  MoveL 782 to (-960, 800, -0.5) mm, rotated rx -180 ry 0 rz 90 deg; joints [11.922, -75.22, 120.913, -51.827, 9.519, 60.758]
  MoveL 783 to (-960, 800, 50) mm, rotated rx 180 ry 0 rz 90 deg; joints [11.922, -77.377, 120.292, -40.937, 11.444, 49.686]
  MoveL 784 to (-960, 850, 50) mm, rotated rx -180 ry 0 rz 90 deg; joints [12.344, -79.438, 122.916, -43.67, 11.235, 52.769]
  MoveL 785 to (-960, 850, -0.5) mm, rotated rx -180 ry 0 rz 90 deg; joints [12.344, -77.191, 123.556, -55.829, 9.358, 65.123]
  MoveL 786 to (-960, 850, 50) mm, rotated rx -180 ry 0 rz 90 deg; joints [12.344, -79.438, 122.916, -43.67, 11.235, 52.769]
  MoveL 787 to (-960, 900, 50) mm, rotated rx 180 ry 0 rz 90 deg; joints [12.796, -81.543, 125.497, -46.231, 11.128, 55.698]
  MoveL 788 to (-960, 900, -0.5) mm, rotated rx 180 ry 0 rz 90 deg; joints [12.796, -79.199, 126.159, -59.572, 9.302, 69.249]
  MoveL 789 to (-960, 900, 50) mm, rotated rx 180 ry 0 rz 90 deg; joints [12.796, -81.543, 125.497, -46.231, 11.128, 55.698]
  MoveL 790 to (-960, 950, 50) mm, rotated rx 180 ry 0 rz 90 deg; joints [13.282, -83.7, 128.037, -48.525, 11.126, 58.38]
  MoveL 791 to (-960, 950, -0.5) mm, rotated rx -180 ry 0 rz 90 deg; joints [13.282, -81.252, 128.723, -62.909, 9.346, 72.993]
  MoveL 792 to (-960, 950, 50) mm, rotated rx 180 ry 0 rz 90 deg; joints [13.282, -83.7, 128.037, -48.525, 11.126, 58.38]
  MoveL 793 to (-960, 1000, 50) mm, rotated rx 180 ry 0 rz 90 deg; joints [13.805, -85.92, 130.536, -50.46, 11.229, 60.727]
  MoveL 794 to (-960, 1000, -0.5) mm, rotated rx -180 ry 0 rz 90 deg; joints [13.805, -83.361, 131.25, -65.713, 9.483, 76.227]
  MoveL 795 to (-960, 1000, 50) mm, rotated rx 180 ry 0 rz 90 deg; joints [13.805, -85.92, 130.536, -50.46, 11.229, 60.727]
  MoveL 796 to (-960, 1050, 50) mm, rotated rx 180 ry 0 rz 90 deg; joints [14.371, -88.215, 132.994, -51.956, 11.439, 62.658]
  MoveL 797 to (-960, 1050, -0.5) mm, rotated rx 180 ry 0 rz 90 deg; joints [14.371, -85.537, 133.739, -67.879, 9.707, 78.851]
  MoveL 798 to (-960, 1050, 50) mm, rotated rx 180 ry 0 rz 90 deg; joints [14.371, -88.215, 132.994, -51.956, 11.439, 62.658]
  MoveL 799 to (-960, 1100, 50) mm, rotated rx 180 ry 0 rz 90 deg; joints [14.983, -90.599, 135.413, -52.948, 11.763, 64.112]
  MoveL 800 to (-960, 1100, -0.5) mm, rotated rx 180 ry 0 rz 90 deg; joints [14.983, -87.793, 136.192, -69.331, 10.015, 80.788]
  MoveL 801 to (-960, 1100, 50) mm, rotated rx 180 ry 0 rz 90 deg; joints [14.983, -90.599, 135.413, -52.948, 11.763, 64.112]
  MoveL 802 to (-960, 1150, 50) mm, rotated rx 180 ry 0 rz 90 deg; joints [15.649, -93.088, 137.79, -53.393, 12.209, 65.046]
  MoveL 803 to (-960, 1150, -0.5) mm, rotated rx 180 ry 0 rz 90 deg; joints [15.649, -90.145, 138.607, -70.016, 10.407, 81.99]
  MoveL 804 to (-960, 1150, 50) mm, rotated rx 180 ry 0 rz 90 deg; joints [15.649, -93.088, 137.79, -53.393, 12.209, 65.046]
  MoveL 805 to (-960, 1200, 50) mm, rotated rx 180 ry 0 rz 90 deg; joints [16.376, -95.702, 140.125, -53.269, 12.79, 65.44]
  MoveL 806 to (-960, 1200, -0.5) mm, rotated rx 180 ry 0 rz 90 deg; joints [16.376, -92.612, 140.985, -69.905, 10.89, 82.431]
  MoveL 807 to (-960, 1200, 50) mm, rotated rx 180 ry 0 rz 90 deg; joints [16.376, -95.702, 140.125, -53.269, 12.79, 65.44]
  MoveL 808 to (-960, 1250, 50) mm, rotated rx 180 ry 0 rz 90 deg; joints [17.171, -98.462, 142.415, -52.579, 13.529, 65.301]
  MoveL 809 to (-960, 1250, -0.5) mm, rotated rx 180 ry 0 rz 90 deg; joints [17.171, -95.217, 143.324, -68.993, 11.479, 82.105]
  MoveL 810 to (-960, 1250, 50) mm, rotated rx 180 ry 0 rz 90 deg; joints [17.171, -98.462, 142.415, -52.579, 13.529, 65.301]
  MoveL 811 to (-960, 1300, 50) mm, rotated rx -180 ry 0 rz 90 deg; joints [18.044, -101.397, 144.658, -51.352, 14.453, 64.657]
  MoveL 812 to (-960, 1300, -0.5) mm, rotated rx -180 ry 0 rz 90 deg; joints [18.044, -97.987, 145.622, -67.292, 12.199, 81.029]
  MoveL 813 to (-960, 1300, 50) mm, rotated rx -180 ry 0 rz 90 deg; joints [18.044, -101.397, 144.658, -51.352, 14.453, 64.657]
  MoveL 814 to (-960, 1350, 50) mm, rotated rx -180 ry 0 rz 90 deg; joints [19.007, -104.538, 146.849, -49.641, 15.603, 63.564]
  MoveL 815 to (-960, 1350, -0.5) mm, rotated rx 180 ry 0 rz 90 deg; joints [19.007, -100.957, 147.875, -64.845, 13.087, 79.247]
  MoveL 816 to (-960, 1350, 50) mm, rotated rx -180 ry 0 rz 90 deg; joints [19.007, -104.538, 146.849, -49.641, 15.603, 63.564]
  MoveL 817 to (-960, 1400, 50) mm, rotated rx -180 ry 0 rz 90 deg; joints [20.075, -107.924, 148.982, -47.525, 17.03, 62.099]
  MoveL 818 to (-960, 1400, -0.5) mm, rotated rx -180 ry 0 rz 90 deg; joints [20.075, -104.168, 150.079, -61.73, 14.198, 76.837]
  MoveL 819 to (-960, 1400, 50) mm, rotated rx -180 ry 0 rz 90 deg; joints [20.075, -107.924, 148.982, -47.525, 17.03, 62.099]
  MoveL 820 to (-960, 1450, 50) mm, rotated rx -180 ry 0 rz 90 deg; joints [21.264, -111.599, 151.05, -45.102, 18.795, 60.359]
  MoveL 821 to (-960, 1450, -0.5) mm, rotated rx 180 ry 0 rz 90 deg; joints [21.264, -107.67, 152.227, -58.062, 15.601, 73.915]
  MoveL 822 to (-960, 1450, 50) mm, rotated rx -180 ry 0 rz 90 deg; joints [21.264, -111.599, 151.05, -45.102, 18.795, 60.359]
  MoveL 823 to (-1030, 50, 50) mm, rotated rx 180 ry 0 rz 90 deg; joints [9.672, -46.591, 72.453, -13.855, 26.202, 20.023]
  MoveL 824 to (-1030, 50, -0.5) mm, rotated rx -180 ry 0 rz 90 deg; joints [9.672, -45.337, 72.996, -14.794, 24.462, 21.062]
  MoveL 825 to (-1030, 50, 50) mm, rotated rx 180 ry 0 rz 90 deg; joints [9.672, -46.591, 72.453, -13.855, 26.202, 20.023]
  MoveL 826 to (-1030, 100, 50) mm, rotated rx 180 ry 0 rz 90 deg; joints [9.896, -48.808, 76.299, -15.015, 24.675, 21.419]
  MoveL 827 to (-1030, 100, -0.5) mm, rotated rx -180 ry 0 rz 90 deg; joints [9.896, -47.51, 76.834, -16.131, 22.91, 22.638]
  MoveL 828 to (-1030, 100, 50) mm, rotated rx 180 ry 0 rz 90 deg; joints [9.896, -48.808, 76.299, -15.015, 24.675, 21.419]
  MoveL 829 to (-1030, 150, 50) mm, rotated rx 180 ry 0 rz 90 deg; joints [10.13, -50.96, 79.988, -16.284, 23.25, 22.928]
  MoveL 830 to (-1030, 150, -0.5) mm, rotated rx 180 ry 0 rz 90 deg; joints [10.13, -49.618, 80.517, -17.61, 21.46, 24.362]
  MoveL 831 to (-1030, 150, 50) mm, rotated rx 180 ry 0 rz 90 deg; joints [10.13, -50.96, 79.988, -16.284, 23.25, 22.928]
  MoveL 832 to (-1030, 200, 50) mm, rotated rx 180 ry 0 rz 90 deg; joints [10.375, -53.058, 83.54, -17.672, 21.922, 24.564]
  MoveL 833 to (-1030, 200, -0.5) mm, rotated rx 180 ry 0 rz 90 deg; joints [10.375, -51.67, 84.065, -19.25, 20.106, 26.254]
  MoveL 834 to (-1030, 200, 50) mm, rotated rx 180 ry 0 rz 90 deg; joints [10.375, -53.058, 83.54, -17.672, 21.922, 24.564]
  MoveL 835 to (-1030, 250, 50) mm, rotated rx 180 ry 0 rz 90 deg; joints [10.632, -55.112, 86.972, -19.192, 20.684, 26.338]
  MoveL 836 to (-1030, 250, -0.5) mm, rotated rx -180 ry 0 rz 90 deg; joints [10.632, -53.676, 87.495, -21.069, 18.844, 28.332]
  MoveL 837 to (-1030, 250, 50) mm, rotated rx 180 ry 0 rz 90 deg; joints [10.632, -55.112, 86.972, -19.192, 20.684, 26.338]
  MoveL 838 to (-1030, 300, 50) mm, rotated rx 180 ry 0 rz 90 deg; joints [10.903, -57.13, 90.296, -20.854, 19.534, 28.262]
  MoveL 839 to (-1030, 300, -0.5) mm, rotated rx -180 ry 0 rz 90 deg; joints [10.903, -55.645, 90.82, -23.087, 17.671, 30.618]
  MoveL 840 to (-1030, 300, 50) mm, rotated rx 180 ry 0 rz 90 deg; joints [10.903, -57.13, 90.296, -20.854, 19.534, 28.262]
  MoveL 841 to (-1030, 350, 50) mm, rotated rx -180 ry 0 rz 90 deg; joints [11.187, -59.119, 93.525, -22.667, 18.471, 30.347]
  MoveL 842 to (-1030, 350, -0.5) mm, rotated rx 180 ry 0 rz 90 deg; joints [11.187, -57.583, 94.051, -25.322, 16.586, 33.131]
  MoveL 843 to (-1030, 350, 50) mm, rotated rx -180 ry 0 rz 90 deg; joints [11.187, -59.119, 93.525, -22.667, 18.471, 30.347]
  MoveL 844 to (-1030, 400, 50) mm, rotated rx -180 ry 0 rz 90 deg; joints [11.486, -61.086, 96.667, -24.639, 17.492, 32.601]
  MoveL 845 to (-1030, 400, -0.5) mm, rotated rx 180 ry 0 rz 90 deg; joints [11.486, -59.497, 97.197, -27.791, 15.591, 35.888]
  MoveL 846 to (-1030, 400, 50) mm, rotated rx -180 ry 0 rz 90 deg; joints [11.486, -61.086, 96.667, -24.639, 17.492, 32.601]
  MoveL 847 to (-1030, 450, 50) mm, rotated rx -180 ry 0 rz 90 deg; joints [11.801, -63.037, 99.73, -26.776, 16.601, 35.03]
  MoveL 848 to (-1030, 450, -0.5) mm, rotated rx -180 ry 0 rz 90 deg; joints [11.801, -61.393, 100.265, -30.507, 14.687, 38.904]
  MoveL 849 to (-1030, 450, 50) mm, rotated rx -180 ry 0 rz 90 deg; joints [11.801, -63.037, 99.73, -26.776, 16.601, 35.03]
  MoveL 850 to (-1030, 500, 50) mm, rotated rx 180 ry 0 rz 90 deg; joints [12.134, -64.977, 102.721, -29.075, 15.796, 37.633]
  MoveL 851 to (-1030, 500, -0.5) mm, rotated rx 180 ry 0 rz 90 deg; joints [12.134, -63.275, 103.263, -33.475, 13.876, 42.184]
  MoveL 852 to (-1030, 500, 50) mm, rotated rx 180 ry 0 rz 90 deg; joints [12.134, -64.977, 102.721, -29.075, 15.796, 37.633]
  MoveL 853 to (-1030, 550, 50) mm, rotated rx 180 ry 0 rz 90 deg; joints [12.486, -66.913, 105.646, -31.528, 15.081, 40.405]
  MoveL 854 to (-1030, 550, -0.5) mm, rotated rx 180 ry 0 rz 90 deg; joints [12.486, -65.149, 106.196, -36.688, 13.163, 45.724]
  MoveL 855 to (-1030, 550, 50) mm, rotated rx 180 ry 0 rz 90 deg; joints [12.486, -66.913, 105.646, -31.528, 15.081, 40.405]
  MoveL 856 to (-1030, 600, 50) mm, rotated rx 180 ry 0 rz 90 deg; joints [12.858, -68.849, 108.509, -34.12, 14.458, 43.328]
  MoveL 857 to (-1030, 600, -0.5) mm, rotated rx 180 ry 0 rz 90 deg; joints [12.858, -67.02, 109.069, -40.125, 12.551, 49.503]
  MoveL 858 to (-1030, 600, 50) mm, rotated rx 180 ry 0 rz 90 deg; joints [12.858, -68.849, 108.509, -34.12, 14.458, 43.328]
  MoveL 859 to (-1030, 650, 50) mm, rotated rx 180 ry 0 rz 90 deg; joints [13.253, -70.791, 111.315, -36.821, 13.93, 46.377]
  MoveL 860 to (-1030, 650, -0.5) mm, rotated rx 180 ry 0 rz 90 deg; joints [13.253, -68.894, 111.886, -43.746, 12.044, 53.482]
  MoveL 861 to (-1030, 650, 50) mm, rotated rx 180 ry 0 rz 90 deg; joints [13.253, -70.791, 111.315, -36.821, 13.93, 46.377]
  MoveL 862 to (-1030, 700, 50) mm, rotated rx 180 ry 0 rz 90 deg; joints [13.673, -72.744, 114.067, -39.592, 13.498, 49.512]
  MoveL 863 to (-1030, 700, -0.5) mm, rotated rx 180 ry 0 rz 90 deg; joints [13.673, -70.774, 114.651, -47.488, 11.643, 57.6]
  MoveL 864 to (-1030, 700, 50) mm, rotated rx 180 ry 0 rz 90 deg; joints [13.673, -72.744, 114.067, -39.592, 13.498, 49.512]
  MoveL 865 to (-1030, 750, 50) mm, rotated rx 180 ry 0 rz 90 deg; joints [14.12, -74.715, 116.768, -42.38, 13.165, 52.682]
  MoveL 866 to (-1030, 750, -0.5) mm, rotated rx -180 ry 0 rz 90 deg; joints [14.12, -72.668, 117.367, -51.27, 11.35, 61.777]
  MoveL 867 to (-1030, 750, 50) mm, rotated rx 180 ry 0 rz 90 deg; joints [14.12, -74.715, 116.768, -42.38, 13.165, 52.682]
  MoveL 868 to (-1030, 800, 50) mm, rotated rx 180 ry 0 rz 90 deg; joints [14.596, -76.709, 119.421, -45.122, 12.932, 55.826]
  MoveL 869 to (-1030, 800, -0.5) mm, rotated rx -180 ry 0 rz 90 deg; joints [14.596, -74.58, 120.037, -54.992, 11.164, 65.916]
  MoveL 870 to (-1030, 800, 50) mm, rotated rx 180 ry 0 rz 90 deg; joints [14.596, -76.709, 119.421, -45.122, 12.932, 55.826]
  MoveL 871 to (-1030, 850, 50) mm, rotated rx 180 ry 0 rz 90 deg; joints [15.104, -78.733, 122.029, -47.746, 12.8, 58.873]
  MoveL 872 to (-1030, 850, -0.5) mm, rotated rx 180 ry 0 rz 90 deg; joints [15.104, -76.517, 122.662, -58.546, 11.083, 69.91]
  MoveL 873 to (-1030, 850, 50) mm, rotated rx 180 ry 0 rz 90 deg; joints [15.104, -78.733, 122.029, -47.746, 12.8, 58.873]
  MoveL 874 to (-1030, 900, 50) mm, rotated rx 180 ry 0 rz 90 deg; joints [15.648, -80.795, 124.591, -50.177, 12.769, 61.751]
  MoveL 875 to (-1030, 900, -0.5) mm, rotated rx 180 ry 0 rz 90 deg; joints [15.648, -78.486, 125.246, -61.823, 11.103, 73.651]
  MoveL 876 to (-1030, 900, 50) mm, rotated rx 180 ry 0 rz 90 deg; joints [15.648, -80.795, 124.591, -50.177, 12.769, 61.751]
  MoveL 877 to (-1030, 950, 50) mm, rotated rx -180 ry 0 rz 90 deg; joints [16.232, -82.903, 127.111, -52.341, 12.839, 64.386]
  MoveL 878 to (-1030, 950, -0.5) mm, rotated rx -180 ry 0 rz 90 deg; joints [16.232, -80.494, 127.788, -64.724, 11.218, 77.043]
  MoveL 879 to (-1030, 950, 50) mm, rotated rx -180 ry 0 rz 90 deg; joints [16.232, -82.903, 127.111, -52.341, 12.839, 64.386]
  MoveL 880 to (-1030, 1000, 50) mm, rotated rx 180 ry 0 rz 90 deg; joints [16.86, -85.066, 129.588, -54.17, 13.01, 66.712]
  MoveL 881 to (-1030, 1000, -0.5) mm, rotated rx 180 ry 0 rz 90 deg; joints [16.86, -82.55, 130.291, -67.162, 11.423, 80.002]
  MoveL 882 to (-1030, 1000, 50) mm, rotated rx 180 ry 0 rz 90 deg; joints [16.86, -85.066, 129.588, -54.17, 13.01, 66.712]
  MoveL 883 to (-1030, 1050, 50) mm, rotated rx 180 ry 0 rz 90 deg; joints [17.536, -87.294, 132.023, -55.605, 13.285, 68.674]
  MoveL 884 to (-1030, 1050, -0.5) mm, rotated rx 180 ry 0 rz 90 deg; joints [17.536, -84.664, 132.755, -69.072, 11.713, 82.464]
  MoveL 885 to (-1030, 1050, 50) mm, rotated rx 180 ry 0 rz 90 deg; joints [17.536, -87.294, 132.023, -55.605, 13.285, 68.674]
  MoveL 886 to (-1030, 1100, 50) mm, rotated rx 180 ry 0 rz 90 deg; joints [18.268, -89.599, 134.415, -56.6, 13.667, 70.228]
  MoveL 887 to (-1030, 1100, -0.5) mm, rotated rx 180 ry 0 rz 90 deg; joints [18.268, -86.847, 135.179, -70.403, 12.087, 84.381]
  MoveL 888 to (-1030, 1100, 50) mm, rotated rx 180 ry 0 rz 90 deg; joints [18.268, -89.599, 134.415, -56.6, 13.667, 70.228]
  MoveL 889 to (-1030, 1150, 50) mm, rotated rx -180 ry 0 rz 90 deg; joints [19.06, -91.995, 136.765, -57.126, 14.164, 71.344]
  MoveL 890 to (-1030, 1150, -0.5) mm, rotated rx -180 ry 0 rz 90 deg; joints [19.06, -89.112, 137.565, -71.123, 12.544, 85.725]
  MoveL 891 to (-1030, 1150, 50) mm, rotated rx -180 ry 0 rz 90 deg; joints [19.06, -91.995, 136.765, -57.126, 14.164, 71.344]
  MoveL 892 to (-1030, 1200, 50) mm, rotated rx -180 ry 0 rz 90 deg; joints [19.922, -94.497, 139.07, -57.164, 14.786, 72.01]
  MoveL 893 to (-1030, 1200, -0.5) mm, rotated rx -180 ry 0 rz 90 deg; joints [19.922, -91.475, 139.91, -71.213, 13.091, 86.479]
  MoveL 894 to (-1030, 1200, 50) mm, rotated rx -180 ry 0 rz 90 deg; joints [19.922, -94.497, 139.07, -57.164, 14.786, 72.01]
  MoveL 895 to (-1100, 50, 50) mm, rotated rx 180 ry 0 rz 90 deg; joints [11.458, -46.001, 71.423, -15.96, 27.042, 23.241]
  MoveL 896 to (-1100, 50, -0.5) mm, rotated rx 180 ry 0 rz 90 deg; joints [11.458, -44.759, 71.968, -16.991, 25.328, 24.39]
  MoveL 897 to (-1100, 50, 50) mm, rotated rx 180 ry 0 rz 90 deg; joints [11.458, -46.001, 71.423, -15.96, 27.042, 23.241]
  MoveL 898 to (-1100, 100, 50) mm, rotated rx 180 ry 0 rz 90 deg; joints [11.72, -48.224, 75.291, -17.252, 25.534, 24.813]
  MoveL 899 to (-1100, 100, -0.5) mm, rotated rx 180 ry 0 rz 90 deg; joints [11.72, -46.938, 75.827, -18.469, 23.799, 26.152]
  MoveL 900 to (-1100, 100, 50) mm, rotated rx 180 ry 0 rz 90 deg; joints [11.72, -48.224, 75.291, -17.252, 25.534, 24.813]
  MoveL 901 to (-1100, 150, 50) mm, rotated rx 180 ry 0 rz 90 deg; joints [11.995, -50.379, 78.996, -18.656, 24.133, 26.501]
  MoveL 902 to (-1100, 150, -0.5) mm, rotated rx -180 ry 0 rz 90 deg; joints [11.995, -49.048, 79.526, -20.092, 22.378, 28.064]
  MoveL 903 to (-1100, 150, 50) mm, rotated rx 180 ry 0 rz 90 deg; joints [11.995, -50.379, 78.996, -18.656, 24.133, 26.501]
  MoveL 904 to (-1100, 200, 50) mm, rotated rx 180 ry 0 rz 90 deg; joints [12.283, -52.477, 82.56, -20.182, 22.834, 28.318]
  MoveL 905 to (-1100, 200, -0.5) mm, rotated rx -180 ry 0 rz 90 deg; joints [12.283, -51.101, 83.086, -21.876, 21.059, 30.144]
  MoveL 906 to (-1100, 200, 50) mm, rotated rx 180 ry 0 rz 90 deg; joints [12.283, -52.477, 82.56, -20.182, 22.834, 28.318]
  MoveL 907 to (-1100, 250, 50) mm, rotated rx -180 ry 0 rz 90 deg; joints [12.585, -54.527, 86, -21.838, 21.63, 30.274]
  MoveL 908 to (-1100, 250, -0.5) mm, rotated rx 180 ry 0 rz 90 deg; joints [12.585, -53.105, 86.523, -23.834, 19.836, 32.408]
  MoveL 909 to (-1100, 250, 50) mm, rotated rx -180 ry 0 rz 90 deg; joints [12.585, -54.527, 86, -21.838, 21.63, 30.274]
  MoveL 910 to (-1100, 300, 50) mm, rotated rx 180 ry 0 rz 90 deg; joints [12.902, -56.54, 89.329, -23.633, 20.519, 32.378]
  MoveL 911 to (-1100, 300, -0.5) mm, rotated rx 180 ry 0 rz 90 deg; joints [12.902, -55.07, 89.853, -25.981, 18.708, 34.87]
  MoveL 912 to (-1100, 300, 50) mm, rotated rx 180 ry 0 rz 90 deg; joints [12.902, -56.54, 89.329, -23.633, 20.519, 32.378]
  MoveL 913 to (-1100, 350, 50) mm, rotated rx 180 ry 0 rz 90 deg; joints [13.234, -58.521, 92.56, -25.572, 19.498, 34.636]
  MoveL 914 to (-1100, 350, -0.5) mm, rotated rx 180 ry 0 rz 90 deg; joints [13.234, -57.001, 93.085, -28.329, 17.674, 37.545]
  MoveL 915 to (-1100, 350, 50) mm, rotated rx 180 ry 0 rz 90 deg; joints [13.234, -58.521, 92.56, -25.572, 19.498, 34.636]
  MoveL 916 to (-1100, 400, 50) mm, rotated rx 180 ry 0 rz 90 deg; joints [13.584, -60.478, 95.701, -27.658, 18.568, 37.054]
  MoveL 917 to (-1100, 400, -0.5) mm, rotated rx 180 ry 0 rz 90 deg; joints [13.584, -58.906, 96.23, -30.887, 16.735, 40.441]
  MoveL 918 to (-1100, 400, 50) mm, rotated rx 180 ry 0 rz 90 deg; joints [13.584, -60.478, 95.701, -27.658, 18.568, 37.054]
  MoveL 919 to (-1100, 450, 50) mm, rotated rx -180 ry 0 rz 90 deg; joints [13.953, -62.416, 98.762, -29.89, 17.728, 39.63]
  MoveL 920 to (-1100, 450, -0.5) mm, rotated rx -180 ry 0 rz 90 deg; joints [13.953, -60.79, 99.295, -33.656, 15.891, 43.562]
  MoveL 921 to (-1100, 450, 50) mm, rotated rx -180 ry 0 rz 90 deg; joints [13.953, -62.416, 98.762, -29.89, 17.728, 39.63]
  MoveL 922 to (-1100, 500, 50) mm, rotated rx -180 ry 0 rz 90 deg; joints [14.342, -64.342, 101.748, -32.262, 16.98, 42.359]
  MoveL 923 to (-1100, 500, -0.5) mm, rotated rx 180 ry 0 rz 90 deg; joints [14.342, -62.659, 102.287, -36.63, 15.146, 46.903]
  MoveL 924 to (-1100, 500, 50) mm, rotated rx -180 ry 0 rz 90 deg; joints [14.342, -64.342, 101.748, -32.262, 16.98, 42.359]
  MoveL 925 to (-1100, 550, 50) mm, rotated rx 180 ry 0 rz 90 deg; joints [14.753, -66.259, 104.665, -34.759, 16.325, 45.228]
  MoveL 926 to (-1100, 550, -0.5) mm, rotated rx 180 ry 0 rz 90 deg; joints [14.753, -64.517, 105.212, -39.791, 14.501, 50.448]
  MoveL 927 to (-1100, 550, 50) mm, rotated rx 180 ry 0 rz 90 deg; joints [14.753, -66.259, 104.665, -34.759, 16.325, 45.228]
  MoveL 928 to (-1100, 600, 50) mm, rotated rx -180 ry 0 rz 90 deg; joints [15.187, -68.175, 107.519, -37.358, 15.765, 48.217]
  MoveL 929 to (-1100, 600, -0.5) mm, rotated rx 180 ry 0 rz 90 deg; joints [15.187, -66.369, 108.076, -43.11, 13.96, 54.167]
  MoveL 930 to (-1100, 600, 50) mm, rotated rx -180 ry 0 rz 90 deg; joints [15.187, -68.175, 107.519, -37.358, 15.765, 48.217]
  MoveL 931 to (-1100, 650, 50) mm, rotated rx -180 ry 0 rz 90 deg; joints [15.647, -70.093, 110.314, -40.029, 15.302, 51.294]
  MoveL 932 to (-1100, 650, -0.5) mm, rotated rx 180 ry 0 rz 90 deg; joints [15.647, -68.221, 110.881, -46.54, 13.523, 58.016]
  MoveL 933 to (-1100, 650, 50) mm, rotated rx -180 ry 0 rz 90 deg; joints [15.647, -70.093, 110.314, -40.029, 15.302, 51.294]
  MoveL 934 to (-1100, 700, 50) mm, rotated rx 180 ry 0 rz 90 deg; joints [16.135, -72.018, 113.053, -42.73, 14.936, 54.421]
  MoveL 935 to (-1100, 700, -0.5) mm, rotated rx 180 ry 0 rz 90 deg; joints [16.135, -70.076, 113.632, -50.021, 13.193, 61.936]
  MoveL 936 to (-1100, 700, 50) mm, rotated rx 180 ry 0 rz 90 deg; joints [16.135, -72.018, 113.053, -42.73, 14.936, 54.421]
  MoveL 937 to (-1100, 750, 50) mm, rotated rx -180 ry 0 rz 90 deg; joints [16.654, -73.957, 115.739, -45.412, 14.67, 57.55]
  MoveL 938 to (-1100, 750, -0.5) mm, rotated rx 180 ry 0 rz 90 deg; joints [16.654, -71.941, 116.332, -53.48, 12.969, 65.857]
  MoveL 939 to (-1100, 750, 50) mm, rotated rx -180 ry 0 rz 90 deg; joints [16.654, -73.957, 115.739, -45.412, 14.67, 57.55]
  MoveL 940 to (-1100, 800, 50) mm, rotated rx 180 ry 0 rz 90 deg; joints [17.206, -75.915, 118.376, -48.019, 14.503, 60.626]
  MoveL 941 to (-1100, 800, -0.5) mm, rotated rx 180 ry 0 rz 90 deg; joints [17.206, -73.82, 118.984, -56.836, 12.849, 69.699]
  MoveL 942 to (-1100, 800, 50) mm, rotated rx 180 ry 0 rz 90 deg; joints [17.206, -75.915, 118.376, -48.019, 14.503, 60.626]
  MoveL 943 to (-1100, 850, 50) mm, rotated rx 180 ry 0 rz 90 deg; joints [17.794, -77.898, 120.964, -50.49, 14.435, 63.591]
  MoveL 944 to (-1100, 850, -0.5) mm, rotated rx 180 ry 0 rz 90 deg; joints [17.794, -75.719, 121.59, -60.007, 12.83, 73.381]
  MoveL 945 to (-1100, 850, 50) mm, rotated rx 180 ry 0 rz 90 deg; joints [17.794, -77.898, 120.964, -50.49, 14.435, 63.591]
  MoveL 946 to (-1100, 900, 50) mm, rotated rx -180 ry 0 rz 90 deg; joints [18.423, -79.912, 123.505, -52.766, 14.466, 66.387]
  MoveL 947 to (-1100, 900, -0.5) mm, rotated rx -180 ry 0 rz 90 deg; joints [18.423, -77.643, 124.151, -62.911, 12.908, 76.826]
  MoveL 948 to (-1100, 900, 50) mm, rotated rx -180 ry 0 rz 90 deg; joints [18.423, -79.912, 123.505, -52.766, 14.466, 66.387]
  MoveL 949 to (-1100, 950, 50) mm, rotated rx -180 ry 0 rz 90 deg; joints [19.096, -81.964, 126.002, -54.789, 14.595, 68.958]
  MoveL 950 to (-1100, 950, -0.5) mm, rotated rx 180 ry 0 rz 90 deg; joints [19.096, -79.6, 126.669, -65.478, 13.079, 79.964]
  MoveL 951 to (-1100, 950, 50) mm, rotated rx -180 ry 0 rz 90 deg; joints [19.096, -81.964, 126.002, -54.789, 14.595, 68.958]
  MoveL 952 to (-1100, 1000, 50) mm, rotated rx 180 ry 0 rz 90 deg; joints [19.819, -84.063, 128.454, -56.508, 14.824, 71.256]
  MoveL 953 to (-1100, 1000, -0.5) mm, rotated rx -180 ry 0 rz 90 deg; joints [19.819, -81.598, 129.145, -67.649, 13.338, 82.739]
  MoveL 954 to (-1100, 1000, 50) mm, rotated rx 180 ry 0 rz 90 deg; joints [19.819, -84.063, 128.454, -56.508, 14.824, 71.256]
  MoveL 955 to (-1100, 1050, 50) mm, rotated rx -180 ry 0 rz 90 deg; joints [20.595, -86.217, 130.861, -57.881, 15.152, 73.241]
  MoveL 956 to (-1100, 1050, -0.5) mm, rotated rx 180 ry 0 rz 90 deg; joints [20.595, -83.643, 131.579, -69.377, 13.682, 85.107]
  MoveL 957 to (-1100, 1050, 50) mm, rotated rx -180 ry 0 rz 90 deg; joints [20.595, -86.217, 130.861, -57.881, 15.152, 73.241]
  MoveL 958 to (-1100, 1100, 50) mm, rotated rx -180 ry 0 rz 90 deg; joints [21.432, -88.435, 133.224, -58.874, 15.582, 74.882]
  MoveL 959 to (-1100, 1100, -0.5) mm, rotated rx -180 ry 0 rz 90 deg; joints [21.432, -85.745, 133.971, -70.629, 14.108, 87.038]
  MoveL 960 to (-1100, 1100, 50) mm, rotated rx -180 ry 0 rz 90 deg; joints [21.432, -88.435, 133.224, -58.874, 15.582, 74.882]
  MoveL 961 to (-1100, 1150, 50) mm, rotated rx 180 ry 0 rz 90 deg; joints [22.336, -90.729, 135.541, -59.466, 16.121, 76.159]
  MoveL 962 to (-1100, 1150, -0.5) mm, rotated rx -180 ry 0 rz 90 deg; joints [22.336, -87.916, 136.322, -71.382, 14.618, 88.512]
  MoveL 963 to (-1100, 1150, 50) mm, rotated rx 180 ry 0 rz 90 deg; joints [22.336, -90.729, 135.541, -59.466, 16.121, 76.159]
  MoveL 964 to (-1100, 1200, 50) mm, rotated rx 180 ry 0 rz 90 deg; joints [23.315, -93.112, 137.812, -59.644, 16.777, 77.064]
  MoveL 965 to (-1100, 1200, -0.5) mm, rotated rx 180 ry 0 rz 90 deg; joints [23.315, -90.167, 138.63, -71.624, 15.216, 89.521]
  MoveL 966 to (-1100, 1200, 50) mm, rotated rx 180 ry 0 rz 90 deg; joints [23.315, -93.112, 137.812, -59.644, 16.777, 77.064]
  MoveL 967 to (-1170, 11.8, 50) mm, rotated rx 180 ry 0 rz 90 deg; joints [13, -43.543, 67.098, -16.852, 29.229, 24.979]
  MoveL 968 to (-1170, 11.8, -0.5) mm, rotated rx 180 ry 0 rz 90 deg; joints [13, -42.347, 67.658, -17.82, 27.554, 26.078]
  MoveL 969 to (-1170, 11.8, 50) mm, rotated rx 180 ry 0 rz 90 deg; joints [13, -43.543, 67.098, -16.852, 29.229, 24.979]
  MoveL 970 to (-1170, 76, 50) mm, rotated rx 180 ry 0 rz 90 deg; joints [13.375, -46.477, 72.254, -18.561, 27.216, 27.095]
  MoveL 971 to (-1170, 76, -0.5) mm, rotated rx 180 ry 0 rz 90 deg; joints [13.375, -45.225, 72.797, -19.749, 25.521, 28.421]
  MoveL 972 to (-1170, 76, 50) mm, rotated rx 180 ry 0 rz 90 deg; joints [13.375, -46.477, 72.254, -18.561, 27.216, 27.095]
  MoveL 973 to (-1170, 140.2, 50) mm, rotated rx -180 ry 0 rz 90 deg; joints [13.772, -49.278, 77.109, -20.444, 25.399, 29.395]
  MoveL 974 to (-1170, 140.2, -0.5) mm, rotated rx 180 ry 0 rz 90 deg; joints [13.772, -47.971, 77.642, -21.9, 23.683, 30.996]
  MoveL 975 to (-1170, 140.2, 50) mm, rotated rx -180 ry 0 rz 90 deg; joints [13.772, -49.278, 77.109, -20.444, 25.399, 29.395]
  MoveL 976 to (-1240, 11.8, 50) mm, rotated rx 180 ry 0 rz 90 deg; joints [14.711, -42.729, 65.657, -18.464, 30.305, 27.613]
  MoveL 977 to (-1240, 11.8, -0.5) mm, rotated rx -180 ry 0 rz 90 deg; joints [14.711, -41.549, 66.222, -19.467, 28.655, 28.765]
  MoveL 978 to (-1240, 11.8, 50) mm, rotated rx 180 ry 0 rz 90 deg; joints [14.711, -42.729, 65.657, -18.464, 30.305, 27.613]
  MoveL 979 to (-1240, 76, 50) mm, rotated rx 180 ry 0 rz 90 deg; joints [15.131, -45.682, 70.864, -20.271, 28.304, 29.881]
  MoveL 980 to (-1240, 76, -0.5) mm, rotated rx 180 ry 0 rz 90 deg; joints [15.131, -44.446, 71.411, -21.493, 26.638, 31.259]
  MoveL 981 to (-1240, 76, 50) mm, rotated rx 180 ry 0 rz 90 deg; joints [15.131, -45.682, 70.864, -20.271, 28.304, 29.881]
  MoveL 982 to (-1240, 140.2, 50) mm, rotated rx 180 ry 0 rz 90 deg; joints [15.576, -48.493, 75.756, -22.246, 26.51, 32.327]
  MoveL 983 to (-1240, 140.2, -0.5) mm, rotated rx 180 ry 0 rz 90 deg; joints [15.576, -47.202, 76.291, -23.73, 24.828, 33.973]
  MoveL 984 to (-1240, 140.2, 50) mm, rotated rx 180 ry 0 rz 90 deg; joints [15.576, -48.493, 75.756, -22.246, 26.51, 32.327]
  MoveL 985 to (-1310, 50, 50) mm, rotated rx 180 ry 0 rz 90 deg; joints [16.668, -43.595, 67.19, -20.975, 30.283, 31.416]
  MoveL 986 to (-1310, 50, -0.5) mm, rotated rx 180 ry 0 rz 90 deg; joints [16.668, -42.399, 67.75, -22.116, 28.65, 32.727]
  MoveL 987 to (-1310, 50, 50) mm, rotated rx 180 ry 0 rz 90 deg; joints [16.668, -43.595, 67.19, -20.975, 30.283, 31.416]
  MoveL 988 to (-1310, 100, 50) mm, rotated rx 180 ry 0 rz 90 deg; joints [17.039, -45.852, 71.162, -22.495, 28.815, 33.339]
  MoveL 989 to (-1310, 100, -0.5) mm, rotated rx -180 ry 0 rz 90 deg; joints [17.039, -44.612, 71.708, -23.815, 27.173, 34.835]
  MoveL 990 to (-1310, 100, 50) mm, rotated rx 180 ry 0 rz 90 deg; joints [17.039, -45.852, 71.162, -22.495, 28.815, 33.339]
  MoveL 991 to (-1310, 150, 50) mm, rotated rx 180 ry 0 rz 90 deg; joints [17.426, -48.025, 74.946, -24.112, 27.473, 35.366]
  MoveL 992 to (-1310, 150, -0.5) mm, rotated rx 180 ry 0 rz 90 deg; joints [17.426, -46.743, 75.483, -25.637, 25.822, 37.072]
  MoveL 993 to (-1310, 150, 50) mm, rotated rx 180 ry 0 rz 90 deg; joints [17.426, -48.025, 74.946, -24.112, 27.473, 35.366]
  MoveL 994 to (-1310, 200, 50) mm, rotated rx 180 ry 0 rz 90 deg; joints [17.83, -50.129, 78.569, -25.831, 26.247, 37.504]
  MoveL 995 to (-1310, 200, -0.5) mm, rotated rx -180 ry 0 rz 90 deg; joints [17.83, -48.804, 79.1, -27.586, 24.589, 39.447]
  MoveL 996 to (-1310, 200, 50) mm, rotated rx 180 ry 0 rz 90 deg; joints [17.83, -50.129, 78.569, -25.831, 26.247, 37.504]
  MoveL 997 to (-1310, 250, 50) mm, rotated rx 180 ry 0 rz 90 deg; joints [18.252, -52.176, 82.052, -27.654, 25.13, 39.755]
  MoveL 998 to (-1310, 250, -0.5) mm, rotated rx -180 ry 0 rz 90 deg; joints [18.252, -50.807, 82.578, -29.668, 23.467, 41.964]
  MoveL 999 to (-1310, 250, 50) mm, rotated rx 180 ry 0 rz 90 deg; joints [18.252, -52.176, 82.052, -27.654, 25.13, 39.755]
  MoveL 1000 to (-1310, 300, 50) mm, rotated rx 180 ry 0 rz 90 deg; joints [18.695, -54.174, 85.41, -29.581, 24.118, 42.121]
  MoveL 1001 to (-1310, 300, -0.5) mm, rotated rx 180 ry 0 rz 90 deg; joints [18.695, -52.76, 85.934, -31.882, 22.452, 44.627]
  MoveL 1002 to (-1310, 300, 50) mm, rotated rx 180 ry 0 rz 90 deg; joints [18.695, -54.174, 85.41, -29.581, 24.118, 42.121]
  MoveL 1003 to (-1310, 350, 50) mm, rotated rx 180 ry 0 rz 90 deg; joints [19.158, -56.132, 88.658, -31.608, 23.208, 44.602]
  MoveL 1004 to (-1310, 350, -0.5) mm, rotated rx 180 ry 0 rz 90 deg; joints [19.158, -54.672, 89.182, -34.227, 21.542, 47.434]
  MoveL 1005 to (-1310, 350, 50) mm, rotated rx 180 ry 0 rz 90 deg; joints [19.158, -56.132, 88.658, -31.608, 23.208, 44.602]
  MoveL 1006 to (-1310, 400, 50) mm, rotated rx 180 ry 0 rz 90 deg; joints [19.645, -58.056, 91.806, -33.728, 22.398, 47.19]
  MoveL 1007 to (-1310, 400, -0.5) mm, rotated rx -180 ry 0 rz 90 deg; joints [19.645, -56.548, 92.33, -36.694, 20.736, 50.379]
  MoveL 1008 to (-1310, 400, 50) mm, rotated rx 180 ry 0 rz 90 deg; joints [19.645, -58.056, 91.806, -33.728, 22.398, 47.19]
  MoveL 1009 to (-1310, 450, 50) mm, rotated rx 180 ry 0 rz 90 deg; joints [20.155, -59.952, 94.862, -35.932, 21.686, 49.878]
  MoveL 1010 to (-1310, 450, -0.5) mm, rotated rx -180 ry 0 rz 90 deg; joints [20.155, -58.394, 95.39, -39.272, 20.033, 53.452]
  MoveL 1011 to (-1310, 450, 50) mm, rotated rx 180 ry 0 rz 90 deg; joints [20.155, -59.952, 94.862, -35.932, 21.686, 49.878]
  MoveL 1012 to (-1310, 500, 50) mm, rotated rx 180 ry 0 rz 90 deg; joints [20.692, -61.826, 97.835, -38.205, 21.072, 52.653]
  MoveL 1013 to (-1310, 500, -0.5) mm, rotated rx -180 ry 0 rz 90 deg; joints [20.692, -60.217, 98.367, -41.942, 19.433, 56.636]
  MoveL 1014 to (-1310, 500, 50) mm, rotated rx 180 ry 0 rz 90 deg; joints [20.692, -61.826, 97.835, -38.205, 21.072, 52.653]
  MoveL 1015 to (-1310, 550, 50) mm, rotated rx -180 ry 0 rz 90 deg; joints [21.257, -63.683, 100.732, -40.527, 20.556, 55.497]
  MoveL 1016 to (-1310, 550, -0.5) mm, rotated rx 180 ry 0 rz 90 deg; joints [21.257, -62.019, 101.269, -44.678, 18.935, 59.906]
  MoveL 1017 to (-1310, 550, 50) mm, rotated rx -180 ry 0 rz 90 deg; joints [21.257, -63.683, 100.732, -40.527, 20.556, 55.497]
  MoveL 1018 to (-1310, 600, 50) mm, rotated rx -180 ry 0 rz 90 deg; joints [21.851, -65.526, 103.557, -42.874, 20.137, 58.387]
  MoveL 1019 to (-1310, 600, -0.5) mm, rotated rx 180 ry 0 rz 90 deg; joints [21.851, -63.807, 104.101, -47.45, 18.539, 63.235]
  MoveL 1020 to (-1310, 600, 50) mm, rotated rx -180 ry 0 rz 90 deg; joints [21.851, -65.526, 103.557, -42.874, 20.137, 58.387]
  MoveL 1021 to (-1310, 650, 50) mm, rotated rx 180 ry 0 rz 90 deg; joints [22.478, -67.361, 106.314, -45.22, 19.814, 61.299]
  MoveL 1022 to (-1310, 650, -0.5) mm, rotated rx 180 ry 0 rz 90 deg; joints [22.478, -65.583, 106.867, -50.222, 18.245, 66.589]
  MoveL 1023 to (-1310, 650, 50) mm, rotated rx 180 ry 0 rz 90 deg; joints [22.478, -67.361, 106.314, -45.22, 19.814, 61.299]
  MoveL 1024 to (-1310, 700, 50) mm, rotated rx -180 ry 0 rz 90 deg; joints [23.141, -69.191, 109.009, -47.534, 19.589, 64.202]
  MoveL 1025 to (-1310, 700, -0.5) mm, rotated rx 180 ry 0 rz 90 deg; joints [23.141, -67.351, 109.571, -52.955, 18.051, 69.928]
  MoveL 1026 to (-1310, 700, 50) mm, rotated rx -180 ry 0 rz 90 deg; joints [23.141, -69.191, 109.009, -47.534, 19.589, 64.202]
  MoveL 1027 to (-1310, 750, 50) mm, rotated rx -180 ry 0 rz 90 deg; joints [23.841, -71.021, 111.644, -49.782, 19.458, 67.067]
  MoveL 1028 to (-1310, 750, -0.5) mm, rotated rx 180 ry 0 rz 90 deg; joints [23.841, -69.116, 112.216, -55.606, 17.955, 73.214]
  MoveL 1029 to (-1310, 750, 50) mm, rotated rx -180 ry 0 rz 90 deg; joints [23.841, -71.021, 111.644, -49.782, 19.458, 67.067]
  MoveL 1030 to (-1310, 800, 50) mm, rotated rx -180 ry 0 rz 90 deg; joints [24.582, -72.855, 114.221, -51.931, 19.423, 69.861]
  MoveL 1031 to (-1310, 800, -0.5) mm, rotated rx -180 ry 0 rz 90 deg; joints [24.582, -70.881, 114.806, -58.133, 17.954, 76.407]
  MoveL 1032 to (-1310, 800, 50) mm, rotated rx -180 ry 0 rz 90 deg; joints [24.582, -72.855, 114.221, -51.931, 19.423, 69.861]
  MoveL 1033 to (-1310, 850, 50) mm, rotated rx -180 ry 0 rz 90 deg; joints [25.367, -74.695, 116.742, -53.947, 19.48, 72.554]
  MoveL 1034 to (-1310, 850, -0.5) mm, rotated rx 180 ry 0 rz 90 deg; joints [25.367, -72.65, 117.341, -60.497, 18.046, 79.47]
  MoveL 1035 to (-1310, 850, 50) mm, rotated rx -180 ry 0 rz 90 deg; joints [25.367, -74.695, 116.742, -53.947, 19.48, 72.554]
  MoveL 1036 to (-1310, 900, 50) mm, rotated rx 180 ry 0 rz 90 deg; joints [26.201, -76.548, 119.21, -55.802, 19.63, 75.118]
  MoveL 1037 to (-1310, 900, -0.5) mm, rotated rx 180 ry 0 rz 90 deg; joints [26.201, -74.426, 119.824, -62.661, 18.228, 82.368]
  MoveL 1038 to (-1310, 900, 50) mm, rotated rx 180 ry 0 rz 90 deg; joints [26.201, -76.548, 119.21, -55.802, 19.63, 75.118]
  MoveL 1039 to (-1310, 950, 50) mm, rotated rx 180 ry 0 rz 90 deg; joints [27.087, -78.415, 121.625, -57.465, 19.871, 77.526]
  MoveL 1040 to (-1310, 950, -0.5) mm, rotated rx 180 ry 0 rz 90 deg; joints [27.087, -76.214, 122.256, -64.594, 18.496, 85.073]
  MoveL 1041 to (-1310, 950, 50) mm, rotated rx 180 ry 0 rz 90 deg; joints [27.087, -78.415, 121.625, -57.465, 19.871, 77.526]
  MoveL 1042 to (-1310, 1000, 50) mm, rotated rx 180 ry 0 rz 90 deg; joints [28.03, -80.303, 123.988, -58.914, 20.202, 79.759]
  MoveL 1043 to (-1310, 1000, -0.5) mm, rotated rx -180 ry 0 rz 90 deg; joints [28.03, -78.016, 124.638, -66.271, 18.848, 87.563]
  MoveL 1044 to (-1310, 1000, 50) mm, rotated rx 180 ry 0 rz 90 deg; joints [28.03, -80.303, 123.988, -58.914, 20.202, 79.759]
  MoveL 1045 to (-1310, 1050, 50) mm, rotated rx 180 ry 0 rz 90 deg; joints [29.036, -82.215, 126.3, -60.13, 20.624, 81.8]
  MoveL 1046 to (-1310, 1050, -0.5) mm, rotated rx 180 ry 0 rz 90 deg; joints [29.036, -79.839, 126.969, -67.671, 19.281, 89.821]
  MoveL 1047 to (-1310, 1050, 50) mm, rotated rx 180 ry 0 rz 90 deg; joints [29.036, -82.215, 126.3, -60.13, 20.624, 81.8]
  MoveL 1048 to (-1310, 1100, 50) mm, rotated rx -180 ry 0 rz 90 deg; joints [30.109, -84.155, 128.559, -61.098, 21.138, 83.637]
  MoveL 1049 to (-1310, 1100, -0.5) mm, rotated rx -180 ry 0 rz 90 deg; joints [30.109, -81.685, 129.251, -68.781, 19.795, 91.836]
  MoveL 1050 to (-1310, 1100, 50) mm, rotated rx -180 ry 0 rz 90 deg; joints [30.109, -84.155, 128.559, -61.098, 21.138, 83.637]
  MoveL 1051 to (-1310, 1150, 50) mm, rotated rx -180 ry 0 rz 90 deg; joints [31.256, -86.129, 130.765, -61.808, 21.745, 85.265]
  MoveL 1052 to (-1310, 1150, -0.5) mm, rotated rx -180 ry 0 rz 90 deg; joints [31.256, -83.559, 131.482, -69.592, 20.389, 93.604]
  MoveL 1053 to (-1310, 1150, 50) mm, rotated rx -180 ry 0 rz 90 deg; joints [31.256, -86.129, 130.765, -61.808, 21.745, 85.265]
  MoveL 1054 to (-1310, 1200, 50) mm, rotated rx 180 ry 0 rz 90 deg; joints [32.484, -88.141, 132.917, -62.258, 22.451, 86.683]
  MoveL 1055 to (-1310, 1200, -0.5) mm, rotated rx -180 ry 0 rz 90 deg; joints [32.484, -85.466, 133.66, -70.1, 21.067, 95.124]
  MoveL 1056 to (-1310, 1200, 50) mm, rotated rx 180 ry 0 rz 90 deg; joints [32.484, -88.141, 132.917, -62.258, 22.451, 86.683]
  MoveL 1057 to (-1380, 50, 50) mm, rotated rx -180 ry 0 rz 90 deg; joints [18.349, -42.572, 65.377, -22.224, 31.586, 33.644]
  MoveL 1058 to (-1380, 50, -0.5) mm, rotated rx 180 ry 0 rz 90 deg; joints [18.349, -41.395, 65.944, -23.358, 29.979, 34.963]
  MoveL 1059 to (-1380, 50, 50) mm, rotated rx -180 ry 0 rz 90 deg; joints [18.349, -42.572, 65.377, -22.224, 31.586, 33.644]
  MoveL 1060 to (-1380, 100, 50) mm, rotated rx -180 ry 0 rz 90 deg; joints [18.751, -44.848, 69.4, -23.773, 30.122, 35.637]
  MoveL 1061 to (-1380, 100, -0.5) mm, rotated rx -180 ry 0 rz 90 deg; joints [18.751, -43.628, 69.952, -25.078, 28.509, 37.133]
  MoveL 1062 to (-1380, 100, 50) mm, rotated rx -180 ry 0 rz 90 deg; joints [18.751, -44.848, 69.4, -23.773, 30.122, 35.637]
  MoveL 1063 to (-1380, 150, 50) mm, rotated rx -180 ry 0 rz 90 deg; joints [19.171, -47.033, 73.225, -25.412, 28.789, 37.725]
  MoveL 1064 to (-1380, 150, -0.5) mm, rotated rx 180 ry 0 rz 90 deg; joints [19.171, -45.771, 73.766, -26.909, 27.171, 39.42]
  MoveL 1065 to (-1380, 150, 50) mm, rotated rx -180 ry 0 rz 90 deg; joints [19.171, -47.033, 73.225, -25.412, 28.789, 37.725]
  MoveL 1066 to (-1380, 200, 50) mm, rotated rx -180 ry 0 rz 90 deg; joints [19.61, -49.144, 76.879, -27.142, 27.579, 39.914]
  MoveL 1067 to (-1380, 200, -0.5) mm, rotated rx -180 ry 0 rz 90 deg; joints [19.61, -47.84, 77.412, -28.853, 25.956, 41.829]
  MoveL 1068 to (-1380, 200, 50) mm, rotated rx -180 ry 0 rz 90 deg; joints [19.61, -49.144, 76.879, -27.142, 27.579, 39.914]
  MoveL 1069 to (-1380, 250, 50) mm, rotated rx 180 ry 0 rz 90 deg; joints [20.068, -51.193, 80.384, -28.964, 26.482, 42.204]
  MoveL 1070 to (-1380, 250, -0.5) mm, rotated rx -180 ry 0 rz 90 deg; joints [20.068, -49.845, 80.912, -30.912, 24.856, 44.365]
  MoveL 1071 to (-1380, 250, 50) mm, rotated rx 180 ry 0 rz 90 deg; joints [20.068, -51.193, 80.384, -28.964, 26.482, 42.204]
  MoveL 1072 to (-1380, 300, 50) mm, rotated rx 180 ry 0 rz 90 deg; joints [20.547, -53.189, 83.759, -30.876, 25.494, 44.596]
  MoveL 1073 to (-1380, 300, -0.5) mm, rotated rx 180 ry 0 rz 90 deg; joints [20.547, -51.797, 84.284, -33.085, 23.868, 47.027]
  MoveL 1074 to (-1380, 300, 50) mm, rotated rx 180 ry 0 rz 90 deg; joints [20.547, -53.189, 83.759, -30.876, 25.494, 44.596]
  MoveL 1075 to (-1380, 350, 50) mm, rotated rx 180 ry 0 rz 90 deg; joints [21.049, -55.14, 87.018, -32.872, 24.61, 47.087]
  MoveL 1076 to (-1380, 350, -0.5) mm, rotated rx 180 ry 0 rz 90 deg; joints [21.049, -53.703, 87.541, -35.366, 22.987, 49.812]
  MoveL 1077 to (-1380, 350, 50) mm, rotated rx 180 ry 0 rz 90 deg; joints [21.049, -55.14, 87.018, -32.872, 24.61, 47.087]
  MoveL 1078 to (-1380, 400, 50) mm, rotated rx 180 ry 0 rz 90 deg; joints [21.574, -57.054, 90.172, -34.946, 23.828, 49.67]
  MoveL 1079 to (-1380, 400, -0.5) mm, rotated rx 180 ry 0 rz 90 deg; joints [21.574, -55.571, 90.696, -37.746, 22.211, 52.712]
  MoveL 1080 to (-1380, 400, 50) mm, rotated rx 180 ry 0 rz 90 deg; joints [21.574, -57.054, 90.172, -34.946, 23.828, 49.67]
  MoveL 1081 to (-1380, 450, 50) mm, rotated rx -180 ry 0 rz 90 deg; joints [22.125, -58.936, 93.23, -37.085, 23.146, 52.335]
  MoveL 1082 to (-1380, 450, -0.5) mm, rotated rx -180 ry 0 rz 90 deg; joints [22.125, -57.405, 93.756, -40.211, 21.539, 55.715]
  MoveL 1083 to (-1380, 450, 50) mm, rotated rx -180 ry 0 rz 90 deg; joints [22.125, -58.936, 93.23, -37.085, 23.146, 52.335]
  MoveL 1084 to (-1380, 500, 50) mm, rotated rx -180 ry 0 rz 90 deg; joints [22.704, -60.793, 96.202, -39.275, 22.563, 55.071]
  MoveL 1085 to (-1380, 500, -0.5) mm, rotated rx -180 ry 0 rz 90 deg; joints [22.704, -59.212, 96.731, -42.743, 20.97, 58.805]
  MoveL 1086 to (-1380, 500, 50) mm, rotated rx -180 ry 0 rz 90 deg; joints [22.704, -60.793, 96.202, -39.275, 22.563, 55.071]
  MoveL 1087 to (-1380, 550, 50) mm, rotated rx -180 ry 0 rz 90 deg; joints [23.311, -62.628, 99.093, -41.498, 22.077, 57.859]
  MoveL 1088 to (-1380, 550, -0.5) mm, rotated rx -180 ry 0 rz 90 deg; joints [23.311, -60.996, 99.626, -45.319, 20.503, 61.959]
  MoveL 1089 to (-1380, 550, 50) mm, rotated rx -180 ry 0 rz 90 deg; joints [23.311, -62.628, 99.093, -41.498, 22.077, 57.859]
  MoveL 1090 to (-1380, 600, 50) mm, rotated rx -180 ry 0 rz 90 deg; joints [23.951, -64.447, 101.909, -43.731, 21.689, 60.68]
  MoveL 1091 to (-1380, 600, -0.5) mm, rotated rx -180 ry 0 rz 90 deg; joints [23.951, -62.76, 102.449, -47.91, 20.136, 65.153]
  MoveL 1092 to (-1380, 600, 50) mm, rotated rx -180 ry 0 rz 90 deg; joints [23.951, -64.447, 101.909, -43.731, 21.689, 60.68]
  MoveL 1093 to (-1380, 650, 50) mm, rotated rx -180 ry 0 rz 90 deg; joints [24.624, -66.252, 104.655, -45.95, 21.397, 63.51]
  MoveL 1094 to (-1380, 650, -0.5) mm, rotated rx 180 ry 0 rz 90 deg; joints [24.624, -64.51, 105.202, -50.486, 19.87, 68.357]
  MoveL 1095 to (-1380, 650, 50) mm, rotated rx -180 ry 0 rz 90 deg; joints [24.624, -66.252, 104.655, -45.95, 21.397, 63.51]
  MoveL 1096 to (-1380, 700, 50) mm, rotated rx -180 ry 0 rz 90 deg; joints [25.333, -68.049, 107.334, -48.129, 21.199, 66.326]
  MoveL 1097 to (-1380, 700, -0.5) mm, rotated rx 180 ry 0 rz 90 deg; joints [25.333, -66.248, 107.89, -53.013, 19.701, 71.538]
  MoveL 1098 to (-1380, 700, 50) mm, rotated rx -180 ry 0 rz 90 deg; joints [25.333, -68.049, 107.334, -48.129, 21.199, 66.326]
  MoveL 1099 to (-1380, 750, 50) mm, rotated rx -180 ry 0 rz 90 deg; joints [26.081, -69.841, 109.951, -50.238, 21.096, 69.101]
  MoveL 1100 to (-1380, 750, -0.5) mm, rotated rx 180 ry 0 rz 90 deg; joints [26.081, -67.978, 110.517, -55.456, 19.627, 74.665]
  MoveL 1101 to (-1380, 750, 50) mm, rotated rx -180 ry 0 rz 90 deg; joints [26.081, -69.841, 109.951, -50.238, 21.096, 69.101]
  MoveL 1102 to (-1380, 800, 50) mm, rotated rx 180 ry 0 rz 90 deg; joints [26.872, -71.631, 112.508, -52.251, 21.085, 71.808]
  MoveL 1103 to (-1380, 800, -0.5) mm, rotated rx 180 ry 0 rz 90 deg; joints [26.872, -69.703, 113.084, -57.781, 19.647, 77.706]
  MoveL 1104 to (-1380, 800, 50) mm, rotated rx 180 ry 0 rz 90 deg; joints [26.872, -71.631, 112.508, -52.251, 21.085, 71.808]
  MoveL 1105 to (-1380, 850, 50) mm, rotated rx -180 ry 0 rz 90 deg; joints [27.708, -73.423, 115.006, -54.14, 21.165, 74.424]
  MoveL 1106 to (-1380, 850, -0.5) mm, rotated rx 180 ry 0 rz 90 deg; joints [27.708, -71.427, 115.595, -59.956, 19.757, 80.63]
  MoveL 1107 to (-1380, 850, 50) mm, rotated rx -180 ry 0 rz 90 deg; joints [27.708, -73.423, 115.006, -54.14, 21.165, 74.424]
  MoveL 1108 to (-1380, 900, 50) mm, rotated rx 180 ry 0 rz 90 deg; joints [28.594, -75.22, 117.448, -55.879, 21.335, 76.924]
  MoveL 1109 to (-1380, 900, -0.5) mm, rotated rx -180 ry 0 rz 90 deg; joints [28.594, -73.153, 118.051, -61.951, 19.955, 83.412]
  MoveL 1110 to (-1380, 900, 50) mm, rotated rx 180 ry 0 rz 90 deg; joints [28.594, -75.22, 117.448, -55.879, 21.335, 76.924]
  MoveL 1111 to (-1380, 950, 50) mm, rotated rx -180 ry 0 rz 90 deg; joints [29.533, -77.025, 119.834, -57.447, 21.594, 79.29]
  MoveL 1112 to (-1380, 950, -0.5) mm, rotated rx 180 ry 0 rz 90 deg; joints [29.533, -74.883, 120.452, -63.742, 20.236, 86.029]
  MoveL 1113 to (-1380, 950, 50) mm, rotated rx -180 ry 0 rz 90 deg; joints [29.533, -77.025, 119.834, -57.447, 21.594, 79.29]
  MoveL 1114 to (-1380, 1000, 50) mm, rotated rx 180 ry 0 rz 90 deg; joints [30.529, -78.842, 122.166, -58.823, 21.94, 81.505]
  MoveL 1115 to (-1380, 1000, -0.5) mm, rotated rx 180 ry 0 rz 90 deg; joints [30.529, -76.621, 122.801, -65.309, 20.6, 88.463]
  MoveL 1116 to (-1380, 1000, 50) mm, rotated rx 180 ry 0 rz 90 deg; joints [30.529, -78.842, 122.166, -58.823, 21.94, 81.505]
  MoveL 1117 to (-1380, 1050, 50) mm, rotated rx -180 ry 0 rz 90 deg; joints [31.588, -80.673, 124.443, -59.994, 22.374, 83.557]
  MoveL 1118 to (-1380, 1050, -0.5) mm, rotated rx -180 ry 0 rz 90 deg; joints [31.588, -78.37, 125.096, -66.635, 21.044, 90.703]
  MoveL 1119 to (-1380, 1050, 50) mm, rotated rx -180 ry 0 rz 90 deg; joints [31.588, -80.673, 124.443, -59.994, 22.374, 83.557]
  MoveL 1120 to (-1380, 1100, 50) mm, rotated rx 180 ry 0 rz 90 deg; joints [32.714, -82.524, 126.665, -60.947, 22.897, 85.437]
  MoveL 1121 to (-1380, 1100, -0.5) mm, rotated rx 180 ry 0 rz 90 deg; joints [32.714, -80.133, 127.338, -67.709, 21.567, 92.739]
  MoveL 1122 to (-1380, 1100, 50) mm, rotated rx 180 ry 0 rz 90 deg; joints [32.714, -82.524, 126.665, -60.947, 22.897, 85.437]
  MoveL 1123 to (-1380, 1150, 50) mm, rotated rx 180 ry 0 rz 90 deg; joints [33.914, -84.395, 128.832, -61.675, 23.509, 87.14]
  MoveL 1124 to (-1380, 1150, -0.5) mm, rotated rx 180 ry 0 rz 90 deg; joints [33.914, -81.913, 129.527, -68.524, 22.168, 94.57]
  MoveL 1125 to (-1380, 1150, 50) mm, rotated rx 180 ry 0 rz 90 deg; joints [33.914, -84.395, 128.832, -61.675, 23.509, 87.14]
  MoveL 1126 to (-1380, 1200, 50) mm, rotated rx 180 ry 0 rz 90 deg; joints [35.194, -86.291, 130.942, -62.175, 24.212, 88.669]
  MoveL 1127 to (-1380, 1200, -0.5) mm, rotated rx -180 ry 0 rz 90 deg; joints [35.194, -83.713, 131.661, -69.078, 22.849, 96.195]
  MoveL 1128 to (-1380, 1200, 50) mm, rotated rx 180 ry 0 rz 90 deg; joints [35.194, -86.291, 130.942, -62.175, 24.212, 88.669]
  MoveL 1129 to (-1450, 50, 50) mm, rotated rx -180 ry 0 rz 90 deg; joints [19.997, -41.432, 63.347, -23.276, 32.997, 35.63]
  MoveL 1130 to (-1450, 50, -0.5) mm, rotated rx -180 ry 0 rz 90 deg; joints [19.997, -40.276, 63.922, -24.387, 31.413, 36.943]
  MoveL 1131 to (-1450, 50, 50) mm, rotated rx -180 ry 0 rz 90 deg; joints [19.997, -41.432, 63.347, -23.276, 32.997, 35.63]
  MoveL 1132 to (-1450, 100, 50) mm, rotated rx -180 ry 0 rz 90 deg; joints [20.429, -43.733, 67.434, -24.84, 31.528, 37.677]
  MoveL 1133 to (-1450, 100, -0.5) mm, rotated rx -180 ry 0 rz 90 deg; joints [20.429, -42.534, 67.992, -26.111, 29.942, 39.156]
  MoveL 1134 to (-1450, 100, 50) mm, rotated rx -180 ry 0 rz 90 deg; joints [20.429, -43.733, 67.434, -24.84, 31.528, 37.677]
  MoveL 1135 to (-1450, 150, 50) mm, rotated rx 180 ry 0 rz 90 deg; joints [20.881, -45.935, 71.308, -26.483, 30.199, 39.809]
  MoveL 1136 to (-1450, 150, -0.5) mm, rotated rx 180 ry 0 rz 90 deg; joints [20.881, -44.694, 71.853, -27.932, 28.61, 41.473]
  MoveL 1137 to (-1450, 150, 50) mm, rotated rx 180 ry 0 rz 90 deg; joints [20.881, -45.935, 71.308, -26.483, 30.199, 39.809]
  MoveL 1138 to (-1450, 200, 50) mm, rotated rx -180 ry 0 rz 90 deg; joints [21.351, -48.056, 74.999, -28.206, 28.998, 42.03]
  MoveL 1139 to (-1450, 200, -0.5) mm, rotated rx -180 ry 0 rz 90 deg; joints [21.351, -46.773, 75.536, -29.853, 27.407, 43.898]
  MoveL 1140 to (-1450, 200, 50) mm, rotated rx -180 ry 0 rz 90 deg; joints [21.351, -48.056, 74.999, -28.206, 28.998, 42.03]
  MoveL 1141 to (-1450, 250, 50) mm, rotated rx -180 ry 0 rz 90 deg; joints [21.842, -50.109, 78.534, -30.009, 27.914, 44.34]
  MoveL 1142 to (-1450, 250, -0.5) mm, rotated rx -180 ry 0 rz 90 deg; joints [21.842, -48.784, 79.064, -31.872, 26.323, 46.433]
  MoveL 1143 to (-1450, 250, 50) mm, rotated rx -180 ry 0 rz 90 deg; joints [21.842, -50.109, 78.534, -30.009, 27.914, 44.34]
  MoveL 1144 to (-1450, 300, 50) mm, rotated rx 180 ry 0 rz 90 deg; joints [22.356, -52.104, 81.93, -31.889, 26.943, 46.739]
  MoveL 1145 to (-1450, 300, -0.5) mm, rotated rx -180 ry 0 rz 90 deg; joints [22.356, -50.737, 82.457, -33.987, 25.354, 49.076]
  MoveL 1146 to (-1450, 300, 50) mm, rotated rx 180 ry 0 rz 90 deg; joints [22.356, -52.104, 81.93, -31.889, 26.943, 46.739]
  MoveL 1147 to (-1450, 350, 50) mm, rotated rx 180 ry 0 rz 90 deg; joints [22.892, -54.051, 85.204, -33.839, 26.079, 49.223]
  MoveL 1148 to (-1450, 350, -0.5) mm, rotated rx -180 ry 0 rz 90 deg; joints [22.892, -52.639, 85.728, -36.19, 24.494, 51.822]
  MoveL 1149 to (-1450, 350, 50) mm, rotated rx 180 ry 0 rz 90 deg; joints [22.892, -54.051, 85.204, -33.839, 26.079, 49.223]
  MoveL 1150 to (-1450, 400, 50) mm, rotated rx -180 ry 0 rz 90 deg; joints [23.454, -55.956, 88.367, -35.851, 25.319, 51.784]
  MoveL 1151 to (-1450, 400, -0.5) mm, rotated rx 180 ry 0 rz 90 deg; joints [23.454, -54.5, 88.891, -38.472, 23.741, 54.664]
  MoveL 1152 to (-1450, 400, 50) mm, rotated rx -180 ry 0 rz 90 deg; joints [23.454, -55.956, 88.367, -35.851, 25.319, 51.784]
  MoveL 1153 to (-1450, 450, 50) mm, rotated rx -180 ry 0 rz 90 deg; joints [24.042, -57.825, 91.431, -37.915, 24.66, 54.413]
  MoveL 1154 to (-1450, 450, -0.5) mm, rotated rx -180 ry 0 rz 90 deg; joints [24.042, -56.323, 91.955, -40.82, 23.093, 57.59]
  MoveL 1155 to (-1450, 450, 50) mm, rotated rx -180 ry 0 rz 90 deg; joints [24.042, -57.825, 91.431, -37.915, 24.66, 54.413]
  MoveL 1156 to (-1450, 500, 50) mm, rotated rx 180 ry 0 rz 90 deg; joints [24.658, -59.665, 94.403, -40.014, 24.101, 57.099]
  MoveL 1157 to (-1450, 500, -0.5) mm, rotated rx -180 ry 0 rz 90 deg; joints [24.658, -58.115, 94.93, -43.214, 22.547, 60.583]
  MoveL 1158 to (-1450, 500, 50) mm, rotated rx 180 ry 0 rz 90 deg; joints [24.658, -59.665, 94.403, -40.014, 24.101, 57.099]
  MoveL 1159 to (-1450, 550, 50) mm, rotated rx -180 ry 0 rz 90 deg; joints [25.305, -61.48, 97.29, -42.133, 23.639, 59.824]
  MoveL 1160 to (-1450, 550, -0.5) mm, rotated rx 180 ry 0 rz 90 deg; joints [25.305, -59.88, 97.821, -45.635, 22.102, 63.624]
  MoveL 1161 to (-1450, 550, 50) mm, rotated rx -180 ry 0 rz 90 deg; joints [25.305, -61.48, 97.29, -42.133, 23.639, 59.824]
  MoveL 1162 to (-1450, 600, 50) mm, rotated rx -180 ry 0 rz 90 deg; joints [25.984, -63.274, 100.099, -44.251, 23.273, 62.571]
  MoveL 1163 to (-1450, 600, -0.5) mm, rotated rx -180 ry 0 rz 90 deg; joints [25.984, -61.623, 100.635, -48.057, 21.757, 66.691]
  MoveL 1164 to (-1450, 600, 50) mm, rotated rx -180 ry 0 rz 90 deg; joints [25.984, -63.274, 100.099, -44.251, 23.273, 62.571]
  MoveL 1165 to (-1450, 650, 50) mm, rotated rx -180 ry 0 rz 90 deg; joints [26.698, -65.051, 102.834, -46.347, 23.003, 65.321]
  MoveL 1166 to (-1450, 650, -0.5) mm, rotated rx 180 ry 0 rz 90 deg; joints [26.698, -63.347, 103.376, -50.454, 21.51, 69.758]
  MoveL 1167 to (-1450, 650, 50) mm, rotated rx -180 ry 0 rz 90 deg; joints [26.698, -65.051, 102.834, -46.347, 23.003, 65.321]
  MoveL 1168 to (-1450, 700, 50) mm, rotated rx -180 ry 0 rz 90 deg; joints [27.449, -66.815, 105.5, -48.397, 22.826, 68.051]
  MoveL 1169 to (-1450, 700, -0.5) mm, rotated rx -180 ry 0 rz 90 deg; joints [27.449, -65.055, 106.049, -52.797, 21.359, 72.799]
  MoveL 1170 to (-1450, 700, 50) mm, rotated rx -180 ry 0 rz 90 deg; joints [27.449, -66.815, 105.5, -48.397, 22.826, 68.051]
  MoveL 1171 to (-1450, 750, 50) mm, rotated rx 180 ry 0 rz 90 deg; joints [28.239, -68.569, 108.1, -50.378, 22.742, 70.741]
  MoveL 1172 to (-1450, 750, -0.5) mm, rotated rx -180 ry 0 rz 90 deg; joints [28.239, -66.75, 108.658, -55.057, 21.3, 75.787]
  MoveL 1173 to (-1450, 750, 50) mm, rotated rx 180 ry 0 rz 90 deg; joints [28.239, -68.569, 108.1, -50.378, 22.742, 70.741]
  MoveL 1174 to (-1450, 800, 50) mm, rotated rx 180 ry 0 rz 90 deg; joints [29.073, -70.317, 110.636, -52.266, 22.748, 73.368]
  MoveL 1175 to (-1450, 800, -0.5) mm, rotated rx 180 ry 0 rz 90 deg; joints [29.073, -68.437, 111.204, -57.206, 21.333, 78.697]
  MoveL 1176 to (-1450, 800, 50) mm, rotated rx 180 ry 0 rz 90 deg; joints [29.073, -70.317, 110.636, -52.266, 22.748, 73.368]
  MoveL 1177 to (-1450, 850, 50) mm, rotated rx -180 ry 0 rz 90 deg; joints [29.953, -72.06, 113.111, -54.039, 22.843, 75.913]
  MoveL 1178 to (-1450, 850, -0.5) mm, rotated rx 180 ry 0 rz 90 deg; joints [29.953, -70.116, 113.691, -59.218, 21.453, 81.504]
  MoveL 1179 to (-1450, 850, 50) mm, rotated rx -180 ry 0 rz 90 deg; joints [29.953, -72.06, 113.111, -54.039, 22.843, 75.913]
  MoveL 1180 to (-1450, 900, 50) mm, rotated rx 180 ry 0 rz 90 deg; joints [30.883, -73.802, 115.527, -55.675, 23.025, 78.357]
  MoveL 1181 to (-1450, 900, -0.5) mm, rotated rx -180 ry 0 rz 90 deg; joints [30.883, -71.792, 116.119, -61.069, 21.659, 84.187]
  MoveL 1182 to (-1450, 900, 50) mm, rotated rx 180 ry 0 rz 90 deg; joints [30.883, -73.802, 115.527, -55.675, 23.025, 78.357]
  MoveL 1183 to (-1450, 950, 50) mm, rotated rx -180 ry 0 rz 90 deg; joints [31.865, -75.546, 117.885, -57.156, 23.294, 80.683]
  MoveL 1184 to (-1450, 950, -0.5) mm, rotated rx 180 ry 0 rz 90 deg; joints [31.865, -73.466, 118.491, -62.738, 21.947, 86.729]
  MoveL 1185 to (-1450, 950, 50) mm, rotated rx -180 ry 0 rz 90 deg; joints [31.865, -75.546, 117.885, -57.156, 23.294, 80.683]
  MoveL 1186 to (-1450, 1000, 50) mm, rotated rx 180 ry 0 rz 90 deg; joints [32.905, -77.295, 120.185, -58.466, 23.648, 82.88]
  MoveL 1187 to (-1450, 1000, -0.5) mm, rotated rx -180 ry 0 rz 90 deg; joints [32.905, -75.141, 120.806, -64.209, 22.315, 89.116]
  MoveL 1188 to (-1450, 1000, 50) mm, rotated rx 180 ry 0 rz 90 deg; joints [32.905, -77.295, 120.185, -58.466, 23.648, 82.88]
  MoveL 1189 to (-1450, 1050, 50) mm, rotated rx 180 ry 0 rz 90 deg; joints [34.007, -79.05, 122.428, -59.594, 24.086, 84.937]
  MoveL 1190 to (-1450, 1050, -0.5) mm, rotated rx 180 ry 0 rz 90 deg; joints [34.007, -76.82, 123.065, -65.469, 22.762, 91.338]
  MoveL 1191 to (-1450, 1050, 50) mm, rotated rx 180 ry 0 rz 90 deg; joints [34.007, -79.05, 122.428, -59.594, 24.086, 84.937]
  MoveL 1192 to (-1450, 1100, 50) mm, rotated rx -180 ry 0 rz 90 deg; joints [35.176, -80.814, 124.614, -60.529, 24.609, 86.847]
  MoveL 1193 to (-1450, 1100, -0.5) mm, rotated rx 180 ry 0 rz 90 deg; joints [35.176, -78.503, 125.268, -66.509, 23.285, 93.388]
  MoveL 1194 to (-1450, 1100, 50) mm, rotated rx -180 ry 0 rz 90 deg; joints [35.176, -80.814, 124.614, -60.529, 24.609, 86.847]
  MoveL 1195 to (-1450, 1150, 50) mm, rotated rx 180 ry 0 rz 90 deg; joints [36.416, -82.588, 126.741, -61.266, 25.217, 88.61]
  MoveL 1196 to (-1450, 1150, -0.5) mm, rotated rx 180 ry 0 rz 90 deg; joints [36.416, -80.194, 127.415, -67.322, 23.885, 95.265]
  MoveL 1197 to (-1450, 1150, 50) mm, rotated rx 180 ry 0 rz 90 deg; joints [36.416, -82.588, 126.741, -61.266, 25.217, 88.61]
  MoveL 1198 to (-1450, 1200, 50) mm, rotated rx -180 ry 0 rz 90 deg; joints [37.733, -84.376, 128.81, -61.802, 25.913, 90.224]
  MoveL 1199 to (-1450, 1200, -0.5) mm, rotated rx 180 ry 0 rz 90 deg; joints [37.733, -81.894, 129.504, -67.906, 24.561, 96.97]
  MoveL 1200 to (-1450, 1200, 50) mm, rotated rx -180 ry 0 rz 90 deg; joints [37.733, -84.376, 128.81, -61.802, 25.913, 90.224]
  MoveL 1201 to (-1520, 53.8, 50) mm, rotated rx 180 ry 0 rz 90 deg; joints [21.645, -40.351, 61.412, -24.262, 34.397, 37.541]
  MoveL 1202 to (-1520, 53.8, -0.5) mm, rotated rx 180 ry 0 rz 90 deg; joints [21.645, -39.214, 61.996, -25.348, 32.835, 38.845]
  MoveL 1203 to (-1520, 53.8, 50) mm, rotated rx 180 ry 0 rz 90 deg; joints [21.645, -40.351, 61.412, -24.262, 34.397, 37.541]
  MoveL 1204 to (-1520, 83.81, 50) mm, rotated rx -180 ry 0 rz 90 deg; joints [21.921, -41.759, 63.93, -25.196, 33.496, 38.788]
  MoveL 1205 to (-1520, 83.81, -0.5) mm, rotated rx -180 ry 0 rz 90 deg; joints [21.921, -40.597, 64.502, -26.37, 31.934, 40.184]
  MoveL 1206 to (-1520, 83.81, 50) mm, rotated rx -180 ry 0 rz 90 deg; joints [21.921, -41.759, 63.93, -25.196, 33.496, 38.788]
  MoveL 1207 to (-1520, 129.48, 50) mm, rotated rx 180 ry 0 rz 90 deg; joints [22.353, -43.825, 67.597, -26.665, 32.23, 40.738]
  MoveL 1208 to (-1520, 129.48, -0.5) mm, rotated rx -180 ry 0 rz 90 deg; joints [22.353, -42.624, 68.154, -27.985, 30.667, 42.285]
  MoveL 1209 to (-1520, 129.48, 50) mm, rotated rx 180 ry 0 rz 90 deg; joints [22.353, -43.825, 67.597, -26.665, 32.23, 40.738]
  MoveL 1210 to (-1520, 159.49, 50) mm, rotated rx 180 ry 0 rz 90 deg; joints [22.645, -45.138, 69.91, -27.662, 31.462, 42.053]
  MoveL 1211 to (-1520, 159.49, -0.5) mm, rotated rx 180 ry 0 rz 90 deg; joints [22.645, -43.912, 70.46, -29.084, 29.899, 43.707]
  MoveL 1212 to (-1520, 159.49, 50) mm, rotated rx 180 ry 0 rz 90 deg; joints [22.645, -45.138, 69.91, -27.662, 31.462, 42.053]
  MoveL 1213 to (-1520, 205.16, 50) mm, rotated rx -180 ry 0 rz 90 deg; joints [23.105, -47.077, 73.301, -29.227, 30.383, 44.109]
  MoveL 1214 to (-1520, 205.16, -0.5) mm, rotated rx 180 ry 0 rz 90 deg; joints [23.105, -45.814, 73.841, -30.816, 28.821, 45.936]
  MoveL 1215 to (-1520, 205.16, 50) mm, rotated rx -180 ry 0 rz 90 deg; joints [23.105, -47.077, 73.301, -29.227, 30.383, 44.109]
  MoveL 1216 to (-1520, 235.17, 50) mm, rotated rx 180 ry 0 rz 90 deg; joints [23.417, -48.318, 75.453, -30.287, 29.73, 45.495]
  MoveL 1217 to (-1520, 235.17, -0.5) mm, rotated rx 180 ry 0 rz 90 deg; joints [23.417, -47.03, 75.989, -31.992, 28.169, 47.443]
  MoveL 1218 to (-1520, 235.17, 50) mm, rotated rx 180 ry 0 rz 90 deg; joints [23.417, -48.318, 75.453, -30.287, 29.73, 45.495]
  MoveL 1219 to (-1520, 280.84, 50) mm, rotated rx -180 ry 0 rz 90 deg; joints [23.907, -50.161, 78.624, -31.945, 28.817, 47.657]
  MoveL 1220 to (-1520, 280.84, -0.5) mm, rotated rx 180 ry 0 rz 90 deg; joints [23.907, -48.835, 79.154, -33.837, 27.258, 49.801]
  MoveL 1221 to (-1520, 280.84, 50) mm, rotated rx -180 ry 0 rz 90 deg; joints [23.907, -50.161, 78.624, -31.945, 28.817, 47.657]
  MoveL 1222 to (-1520, 310.85, 50) mm, rotated rx -180 ry 0 rz 90 deg; joints [24.24, -51.346, 80.645, -33.062, 28.268, 49.111]
  MoveL 1223 to (-1520, 310.85, -0.5) mm, rotated rx 180 ry 0 rz 90 deg; joints [24.24, -49.995, 81.173, -35.085, 26.712, 51.392]
  MoveL 1224 to (-1520, 310.85, 50) mm, rotated rx -180 ry 0 rz 90 deg; joints [24.24, -51.346, 80.645, -33.062, 28.268, 49.111]
  MoveL 1225 to (-1520, 356.52, 50) mm, rotated rx 180 ry 0 rz 90 deg; joints [24.763, -53.114, 83.634, -34.8, 27.508, 51.373]
  MoveL 1226 to (-1520, 356.52, -0.5) mm, rotated rx 180 ry 0 rz 90 deg; joints [24.763, -51.724, 84.159, -37.03, 25.957, 53.87]
  MoveL 1227 to (-1520, 356.52, 50) mm, rotated rx 180 ry 0 rz 90 deg; joints [24.763, -53.114, 83.634, -34.8, 27.508, 51.373]
  MoveL 1228 to (-1520, 386.53, 50) mm, rotated rx -180 ry 0 rz 90 deg; joints [25.118, -54.255, 85.545, -35.965, 27.057, 52.889]
  MoveL 1229 to (-1520, 386.53, -0.5) mm, rotated rx -180 ry 0 rz 90 deg; joints [25.118, -52.839, 86.069, -38.337, 25.51, 55.535]
  MoveL 1230 to (-1520, 386.53, 50) mm, rotated rx -180 ry 0 rz 90 deg; joints [25.118, -54.255, 85.545, -35.965, 27.057, 52.889]
  MoveL 1231 to (-1690.15, 68.53, 50) mm, rotated rx 180 ry 0 rz 90 deg; joints [25.576, -37.452, 56.186, -26.137, 38.078, 41.523]
  MoveL 1232 to (-1690.15, 68.53, -0.5) mm, rotated rx 180 ry 0 rz 90 deg; joints [25.576, -36.368, 56.8, -27.136, 36.559, 42.779]
  MoveL 1233 to (-1690.15, 68.53, 50) mm, rotated rx 180 ry 0 rz 90 deg; joints [25.576, -37.452, 56.186, -26.137, 38.078, 41.523]
  MoveL 1234 to (-1690.15, 118.53, 50) mm, rotated rx -180 ry 0 rz 90 deg; joints [26.105, -39.851, 60.515, -27.687, 36.581, 43.695]
  MoveL 1235 to (-1690.15, 118.53, -0.5) mm, rotated rx -180 ry 0 rz 90 deg; joints [26.105, -38.724, 61.104, -28.812, 35.069, 45.083]
  MoveL 1236 to (-1690.15, 118.53, 50) mm, rotated rx -180 ry 0 rz 90 deg; joints [26.105, -39.851, 60.515, -27.687, 36.581, 43.695]
  MoveL 1237 to (-1690.15, 168.53, 50) mm, rotated rx 180 ry 0 rz 90 deg; joints [26.653, -42.119, 64.571, -29.282, 35.253, 45.914]
  MoveL 1238 to (-1690.15, 168.53, -0.5) mm, rotated rx -180 ry 0 rz 90 deg; joints [26.653, -40.95, 65.14, -30.544, 33.746, 47.444]
  MoveL 1239 to (-1690.15, 168.53, 50) mm, rotated rx 180 ry 0 rz 90 deg; joints [26.653, -42.119, 64.571, -29.282, 35.253, 45.914]
  MoveL 1240 to (-1690.15, 271.33, 50) mm, rotated rx 180 ry 0 rz 90 deg; joints [27.852, -46.463, 72.23, -32.699, 32.973, 50.63]
  MoveL 1241 to (-1690.15, 271.33, -0.5) mm, rotated rx 180 ry 0 rz 90 deg; joints [27.852, -45.212, 72.773, -34.27, 31.476, 52.487]
  MoveL 1242 to (-1690.15, 271.33, 50) mm, rotated rx 180 ry 0 rz 90 deg; joints [27.852, -46.463, 72.23, -32.699, 32.973, 50.63]
  MoveL 1243 to (-1690.15, 321.33, 50) mm, rotated rx -180 ry 0 rz 90 deg; joints [28.471, -48.453, 75.687, -34.419, 32.057, 52.998]
  MoveL 1244 to (-1690.15, 321.33, -0.5) mm, rotated rx -180 ry 0 rz 90 deg; joints [28.471, -47.163, 76.222, -36.153, 30.566, 55.027]
  MoveL 1245 to (-1690.15, 321.33, 50) mm, rotated rx -180 ry 0 rz 90 deg; joints [28.471, -48.453, 75.687, -34.419, 32.057, 52.998]
  MoveL 1246 to (-1690.15, 371.33, 50) mm, rotated rx -180 ry 0 rz 90 deg; joints [29.116, -50.38, 78.998, -36.169, 31.256, 55.408]
  MoveL 1247 to (-1690.15, 371.33, -0.5) mm, rotated rx -180 ry 0 rz 90 deg; joints [29.116, -49.05, 79.528, -38.074, 29.773, 57.619]
  MoveL 1248 to (-1690.15, 371.33, 50) mm, rotated rx -180 ry 0 rz 90 deg; joints [29.116, -50.38, 78.998, -36.169, 31.256, 55.408]
  MoveL 1249 to (-1566.88, 10, 50) mm, rotated rx 180 ry 0 rz 90 deg; joints [22.303, -37.261, 55.839, -23.428, 36.918, 36.789]
  MoveL 1250 to (-1566.88, 10, -0.5) mm, rotated rx 180 ry 0 rz 90 deg; joints [22.303, -36.18, 56.456, -24.37, 35.366, 37.955]
  MoveL 1251 to (-1566.88, 10, 50) mm, rotated rx 180 ry 0 rz 90 deg; joints [22.303, -37.261, 55.839, -23.428, 36.918, 36.789]
  MoveL 1252 to (-1605.08, 10, 50) mm, rotated rx 180 ry 0 rz 90 deg; joints [23.145, -36.439, 54.345, -23.772, 37.853, 37.554]
  MoveL 1253 to (-1605.08, 10, -0.5) mm, rotated rx -180 ry 0 rz 90 deg; joints [23.145, -35.373, 54.972, -24.691, 36.31, 38.706]
  MoveL 1254 to (-1605.08, 10, 50) mm, rotated rx 180 ry 0 rz 90 deg; joints [23.145, -36.439, 54.345, -23.772, 37.853, 37.554]
  MoveL 1255 to (-1643.28, 10, 50) mm, rotated rx 180 ry 0 rz 90 deg; joints [23.977, -35.569, 52.76, -24.071, 38.829, 38.255]
  MoveL 1256 to (-1643.28, 10, -0.5) mm, rotated rx 180 ry 0 rz 90 deg; joints [23.977, -34.519, 53.399, -24.966, 37.292, 39.391]
  MoveL 1257 to (-1643.28, 10, 50) mm, rotated rx 180 ry 0 rz 90 deg; joints [23.977, -35.569, 52.76, -24.071, 38.829, 38.255]
  MoveL 1258 to (-1566.88, 430, 50) mm, rotated rx -180 ry 0 rz 90 deg; joints [26.857, -55.025, 86.828, -37.946, 27.538, 56.142]
  MoveL 1259 to (-1566.88, 430, -0.5) mm, rotated rx 180 ry 0 rz 90 deg; joints [26.857, -53.591, 87.351, -40.396, 26.02, 58.886]
  MoveL 1260 to (-1566.88, 430, 50) mm, rotated rx -180 ry 0 rz 90 deg; joints [26.857, -55.025, 86.828, -37.946, 27.538, 56.142]
  MoveL 1261 to (-1605.08, 430, 50) mm, rotated rx 180 ry 0 rz 90 deg; joints [27.821, -54.296, 85.614, -38.098, 28.426, 56.886]
  MoveL 1262 to (-1605.08, 430, -0.5) mm, rotated rx -180 ry 0 rz 90 deg; joints [27.821, -52.879, 86.138, -40.441, 26.923, 59.531]
  MoveL 1263 to (-1605.08, 430, 50) mm, rotated rx 180 ry 0 rz 90 deg; joints [27.821, -54.296, 85.614, -38.098, 28.426, 56.886]
  MoveL 1264 to (-1643.28, 430, 50) mm, rotated rx -180 ry 0 rz 90 deg; joints [28.769, -53.539, 84.347, -38.196, 29.328, 57.555]
  MoveL 1265 to (-1643.28, 430, -0.5) mm, rotated rx -180 ry 0 rz 90 deg; joints [28.769, -52.139, 84.872, -40.433, 27.839, 60.103]
  MoveL 1266 to (-1643.28, 430, 50) mm, rotated rx -180 ry 0 rz 90 deg; joints [28.769, -53.539, 84.347, -38.196, 29.328, 57.555]
  MoveL 1267 to (-1520, 821.53, 50) mm, rotated rx -180 ry 0 rz 90 deg; joints [31.573, -69.648, 109.672, -52.778, 24.443, 75.686]
  MoveL 1268 to (-1520, 821.53, -0.5) mm, rotated rx -180 ry 0 rz 90 deg; joints [31.573, -67.792, 110.236, -57.288, 23.055, 80.613]
  MoveL 1269 to (-1520, 821.53, 50) mm, rotated rx -180 ry 0 rz 90 deg; joints [31.573, -69.648, 109.672, -52.778, 24.443, 75.686]
  MoveL 1270 to (-1520, 876.86, 50) mm, rotated rx 180 ry 0 rz 90 deg; joints [32.613, -71.522, 112.353, -54.558, 24.603, 78.384]
  MoveL 1271 to (-1520, 876.86, -0.5) mm, rotated rx 180 ry 0 rz 90 deg; joints [32.613, -69.598, 112.929, -59.282, 23.237, 83.551]
  MoveL 1272 to (-1520, 876.86, 50) mm, rotated rx 180 ry 0 rz 90 deg; joints [32.613, -71.522, 112.353, -54.558, 24.603, 78.384]
  MoveL 1273 to (-1520, 947.66, 50) mm, rotated rx 180 ry 0 rz 90 deg; joints [34.037, -73.91, 115.675, -56.595, 24.958, 81.663]
  MoveL 1274 to (-1520, 947.66, -0.5) mm, rotated rx -180 ry 0 rz 90 deg; joints [34.037, -71.895, 116.267, -61.554, 23.616, 87.102]
  MoveL 1275 to (-1520, 947.66, 50) mm, rotated rx 180 ry 0 rz 90 deg; joints [34.037, -73.91, 115.675, -56.595, 24.958, 81.663]
  MoveL 1276 to (-1520, 1003, 50) mm, rotated rx 180 ry 0 rz 90 deg; joints [35.227, -75.772, 118.186, -57.977, 25.35, 84.071]
  MoveL 1277 to (-1520, 1003, -0.5) mm, rotated rx -180 ry 0 rz 90 deg; joints [35.227, -73.683, 118.793, -63.088, 24.022, 89.694]
  MoveL 1278 to (-1520, 1003, 50) mm, rotated rx 180 ry 0 rz 90 deg; joints [35.227, -75.772, 118.186, -57.977, 25.35, 84.071]
  MoveL 1279 to (-1520, 1073.8, 50) mm, rotated rx 180 ry 0 rz 90 deg; joints [36.859, -78.154, 121.292, -59.451, 25.998, 86.936]
  MoveL 1280 to (-1520, 1073.8, -0.5) mm, rotated rx 180 ry 0 rz 90 deg; joints [36.859, -75.964, 121.92, -64.714, 24.677, 92.758]
  MoveL 1281 to (-1520, 1073.8, 50) mm, rotated rx 180 ry 0 rz 90 deg; joints [36.859, -78.154, 121.292, -59.451, 25.998, 86.936]
  MoveL 1282 to (-1520, 1129.13, 50) mm, rotated rx 180 ry 0 rz 90 deg; joints [38.228, -80.017, 123.636, -60.361, 26.618, 88.999]
  MoveL 1283 to (-1520, 1129.13, -0.5) mm, rotated rx 180 ry 0 rz 90 deg; joints [38.228, -77.744, 124.282, -65.71, 25.292, 94.947]
  MoveL 1284 to (-1520, 1129.13, 50) mm, rotated rx 180 ry 0 rz 90 deg; joints [38.228, -80.017, 123.636, -60.361, 26.618, 88.999]
  MoveL 1285 to (-1690.15, 824.48, 50) mm, rotated rx 180 ry 0 rz 90 deg; joints [36.416, -65.966, 104.222, -51.546, 28.494, 77.726]
  MoveL 1286 to (-1690.15, 824.48, -0.5) mm, rotated rx 180 ry 0 rz 90 deg; joints [36.416, -64.232, 104.768, -55.01, 27.13, 81.642]
  MoveL 1287 to (-1690.15, 824.48, 50) mm, rotated rx 180 ry 0 rz 90 deg; joints [36.416, -65.966, 104.222, -51.546, 28.494, 77.726]
  MoveL 1288 to (-1690.15, 874.48, 50) mm, rotated rx 180 ry 0 rz 90 deg; joints [37.42, -67.55, 106.595, -52.947, 28.631, 80.033]
  MoveL 1289 to (-1690.15, 874.48, -0.5) mm, rotated rx 180 ry 0 rz 90 deg; joints [37.42, -65.765, 107.148, -56.545, 27.28, 84.106]
  MoveL 1290 to (-1690.15, 874.48, 50) mm, rotated rx 180 ry 0 rz 90 deg; joints [37.42, -67.55, 106.595, -52.947, 28.631, 80.033]
  MoveL 1291 to (-1690.15, 924.48, 50) mm, rotated rx 180 ry 0 rz 90 deg; joints [38.471, -69.116, 108.899, -54.241, 28.846, 82.271]
  MoveL 1292 to (-1690.15, 924.48, -0.5) mm, rotated rx 180 ry 0 rz 90 deg; joints [38.471, -67.278, 109.46, -57.96, 27.507, 86.489]
  MoveL 1293 to (-1690.15, 924.48, 50) mm, rotated rx 180 ry 0 rz 90 deg; joints [38.471, -69.116, 108.899, -54.241, 28.846, 82.271]
  MoveL 1294 to (-1690.15, 974.48, 50) mm, rotated rx 180 ry 0 rz 90 deg; joints [39.573, -70.665, 111.135, -55.421, 29.139, 84.432]
  MoveL 1295 to (-1690.15, 974.48, -0.5) mm, rotated rx 180 ry 0 rz 90 deg; joints [39.573, -68.773, 111.706, -59.245, 27.809, 88.781]
  MoveL 1296 to (-1690.15, 974.48, 50) mm, rotated rx 180 ry 0 rz 90 deg; joints [39.573, -70.665, 111.135, -55.421, 29.139, 84.432]
  MoveL 1297 to (-1690.15, 1024.47, 50) mm, rotated rx -180 ry 0 rz 90 deg; joints [40.729, -72.198, 113.304, -56.477, 29.508, 86.509]
  MoveL 1298 to (-1690.15, 1024.47, -0.5) mm, rotated rx -180 ry 0 rz 90 deg; joints [40.729, -70.249, 113.885, -60.391, 28.183, 90.977]
  MoveL 1299 to (-1690.15, 1024.47, 50) mm, rotated rx -180 ry 0 rz 90 deg; joints [40.729, -72.198, 113.304, -56.477, 29.508, 86.509]
  MoveL 1300 to (-1690.15, 1074.47, 50) mm, rotated rx 180 ry 0 rz 90 deg; joints [41.942, -73.715, 115.408, -57.404, 29.951, 88.5]
  MoveL 1301 to (-1690.15, 1074.47, -0.5) mm, rotated rx 180 ry 0 rz 90 deg; joints [41.942, -71.708, 115.999, -61.392, 28.628, 93.072]
  MoveL 1302 to (-1690.15, 1074.47, 50) mm, rotated rx 180 ry 0 rz 90 deg; joints [41.942, -73.715, 115.408, -57.404, 29.951, 88.5]
  MoveL 1303 to (-1690.15, 1124.47, 50) mm, rotated rx 180 ry 0 rz 90 deg; joints [43.215, -75.217, 117.445, -58.196, 30.467, 90.402]
  MoveL 1304 to (-1690.15, 1124.47, -0.5) mm, rotated rx -180 ry 0 rz 90 deg; joints [43.215, -73.15, 118.047, -62.243, 29.14, 95.065]
  MoveL 1305 to (-1690.15, 1124.47, 50) mm, rotated rx 180 ry 0 rz 90 deg; joints [43.215, -75.217, 117.445, -58.196, 30.467, 90.402]
  MoveL 1306 to (-1566.88, 763, 50) mm, rotated rx 180 ry 0 rz 90 deg; joints [31.883, -66.692, 105.315, -50.542, 25.501, 73.436]
  MoveL 1307 to (-1566.88, 763, -0.5) mm, rotated rx -180 ry 0 rz 90 deg; joints [31.883, -64.935, 105.864, -54.503, 24.097, 77.799]
  MoveL 1308 to (-1566.88, 763, 50) mm, rotated rx 180 ry 0 rz 90 deg; joints [31.883, -66.692, 105.315, -50.542, 25.501, 73.436]
  MoveL 1309 to (-1605.08, 763, 50) mm, rotated rx 180 ry 0 rz 90 deg; joints [32.953, -65.881, 104.094, -50.324, 26.408, 73.934]
  MoveL 1310 to (-1605.08, 763, -0.5) mm, rotated rx 180 ry 0 rz 90 deg; joints [32.953, -64.15, 104.639, -54.06, 25.012, 78.08]
  MoveL 1311 to (-1605.08, 763, 50) mm, rotated rx 180 ry 0 rz 90 deg; joints [32.953, -65.881, 104.094, -50.324, 26.408, 73.934]
  MoveL 1312 to (-1643.28, 763, 50) mm, rotated rx -180 ry 0 rz 90 deg; joints [33.998, -65.046, 102.826, -50.064, 27.318, 74.363]
  MoveL 1313 to (-1643.28, 763, -0.5) mm, rotated rx -180 ry 0 rz 90 deg; joints [33.998, -63.341, 103.368, -53.589, 25.929, 78.305]
  MoveL 1314 to (-1643.28, 763, 50) mm, rotated rx -180 ry 0 rz 90 deg; joints [33.998, -65.046, 102.826, -50.064, 27.318, 74.363]
  MoveL 1315 to (-1566.88, 1183, 50) mm, rotated rx -180 ry 0 rz 90 deg; joints [41.146, -80.513, 124.246, -60.536, 28.398, 91.469]
  MoveL 1316 to (-1566.88, 1183, -0.5) mm, rotated rx -180 ry 0 rz 90 deg; joints [41.146, -78.216, 124.897, -65.537, 27.059, 97.117]
  MoveL 1317 to (-1566.88, 1183, 50) mm, rotated rx -180 ry 0 rz 90 deg; joints [41.146, -80.513, 124.246, -60.536, 28.398, 91.469]
  MoveL 1318 to (-1605.08, 1183, 50) mm, rotated rx -180 ry 0 rz 90 deg; joints [42.32, -79.423, 122.896, -60.082, 29.265, 91.874]
  MoveL 1319 to (-1605.08, 1183, -0.5) mm, rotated rx -180 ry 0 rz 90 deg; joints [42.32, -77.176, 123.537, -64.779, 27.927, 97.223]
  MoveL 1320 to (-1605.08, 1183, 50) mm, rotated rx -180 ry 0 rz 90 deg; joints [42.32, -79.423, 122.896, -60.082, 29.265, 91.874]
  MoveL 1321 to (-1643.28, 1183, 50) mm, rotated rx 180 ry 0 rz 90 deg; joints [43.452, -78.321, 121.505, -59.592, 30.122, 92.204]
  MoveL 1322 to (-1643.28, 1183, -0.5) mm, rotated rx -180 ry 0 rz 90 deg; joints [43.452, -76.123, 122.135, -64.007, 28.785, 97.273]
  MoveL 1323 to (-1643.28, 1183, 50) mm, rotated rx 180 ry 0 rz 90 deg; joints [43.452, -78.321, 121.505, -59.592, 30.122, 92.204]
  Set speed (1000.0 mm/s)
  MoveL 1324 to (-1643.28, 1183, 50) mm, rotated rx 180 ry 0 rz 90 deg; joints [43.452, -78.321, 121.505, -59.592, 30.122, 92.204]
  MoveL 1325 to (-1643.28, 1183, 150) mm, rotated rx 180 ry 0 rz 90 deg; joints [43.452, -82.309, 119.903, -52.09, 33.269, 83.396]
